LIN {X 0.075,Y -335.216,Z 1636.671,A 0.000,B 0.000,C 90.000,E1 120.797} C_DIS
LIN {X -0.094,Y -338.872,Z 1636.669,A 0.000,B 0.000,C 90.000,E1 120.384} C_DIS
LIN {X 0.042,Y -340.680,Z 1636.667,A 0.000,B 0.000,C 90.000,E1 120.050} C_DIS
LIN {X 0.186,Y -357.152,Z 1636.647,A 0.000,B 0.000,C 90.000,E1 116.360} C_DIS
LIN {X 0.077,Y -371.127,Z 1636.632,A 0.000,B 0.000,C 90.000,E1 113.695} C_DIS
LIN {X 0.128,Y -384.896,Z 1636.619,A 0.000,B 0.000,C 90.000,E1 111.354} C_DIS
LIN {X 0.030,Y -400.035,Z 1636.606,A 0.000,B 0.000,C 90.000,E1 109.087} C_DIS
LIN {X 0.035,Y -416.645,Z 1636.594,A 0.000,B 0.000,C 90.000,E1 106.858} C_DIS
LIN {X -0.200,Y -434.843,Z 1636.582,A 0.000,B 0.000,C 90.000,E1 104.717} C_DIS
LIN {X 0.091,Y -454.503,Z 1636.570,A 0.000,B 0.000,C 90.000,E1 102.591} C_DIS
LIN {X 0.158,Y -474.801,Z 1636.559,A 0.000,B 0.000,C 90.000,E1 100.658} C_DIS
LIN {X 0.135,Y -498.204,Z 1636.548,A 0.000,B 0.000,C 90.000,E1 98.681} C_DIS
LIN {X -0.215,Y -500.316,Z 1636.547,A 0.000,B 0.000,C 90.000,E1 98.511} C_DIS
LIN {X 0.233,Y -502.133,Z 1636.546,A 0.000,B 0.000,C 90.000,E1 98.219} C_DIS
LIN {X 0.114,Y -503.496,Z 1636.544,A 0.000,B 0.000,C 90.000,E1 97.992} C_DIS
LIN {X -0.087,Y -505.220,Z 1636.542,A 0.000,B 0.000,C 90.000,E1 97.530} C_DIS
LIN {X -0.279,Y -505.833,Z 1636.539,A 0.000,B 0.000,C 90.000,E1 97.068} C_DIS
LIN {X 0.041,Y -505.440,Z 1636.536,A 0.000,B 0.000,C 90.000,E1 96.549} C_DIS
LIN {X -0.139,Y -503.977,Z 1636.534,A 0.000,B 0.000,C 90.000,E1 96.087} C_DIS
LIN {X -0.204,Y -502.765,Z 1636.532,A 0.000,B 0.000,C 90.000,E1 95.853} C_DIS
LIN {X 0.120,Y -492.693,Z 1636.524,A 0.000,B 0.000,C 90.000,E1 94.359} C_DIS
LIN {X -0.215,Y -482.497,Z 1636.516,A 0.000,B 0.000,C 90.000,E1 92.922} C_DIS
LIN {X 0.208,Y -472.061,Z 1636.508,A 0.000,B 0.000,C 90.000,E1 91.375} C_DIS
LIN {X -0.031,Y -461.326,Z 1636.499,A 0.000,B 0.000,C 90.000,E1 89.885} C_DIS
LIN {X 0.010,Y -450.327,Z 1636.491,A 0.000,B 0.000,C 90.000,E1 88.339} C_DIS
LIN {X 0.132,Y -440.740,Z 1636.484,A 0.000,B 0.000,C 90.000,E1 87.020} C_DIS
LIN {X -0.147,Y -428.850,Z 1636.475,A 0.000,B 0.000,C 90.000,E1 85.469} C_DIS
LIN {X 0.070,Y -413.097,Z 1636.463,A 0.000,B 0.000,C 90.000,E1 83.280} C_DIS
LIN {X -0.188,Y -390.844,Z 1636.444,A 0.000,B 0.000,C 90.000,E1 79.982} C_DIS
LIN {X -0.184,Y -373.709,Z 1636.428,A 0.000,B 0.000,C 90.000,E1 77.117} C_DIS
LIN {X -0.093,Y -360.590,Z 1636.415,A 0.000,B 0.000,C 90.000,E1 74.755} C_DIS
LIN {X -0.182,Y -344.772,Z 1636.399,A 0.000,B 0.000,C 90.000,E1 71.764} C_DIS
LIN {X 0.065,Y -334.278,Z 1636.387,A 0.000,B 0.000,C 90.000,E1 69.571} C_DIS
LIN {X 0.131,Y -318.411,Z 1636.367,A 0.000,B 0.000,C 90.000,E1 66.102} C_DIS
LIN {X -0.065,Y -307.744,Z 1636.353,A 0.000,B 0.000,C 90.000,E1 63.563} C_DIS
LIN {X 0.008,Y -298.459,Z 1636.340,A 0.000,B 0.000,C 90.000,E1 61.257} C_DIS
LIN {X -0.096,Y -290.364,Z 1636.329,A 0.000,B 0.000,C 90.000,E1 59.282} C_DIS
LIN {X -0.050,Y -282.053,Z 1636.318,A 0.000,B 0.000,C 90.000,E1 57.248} C_DIS
LIN {X 0.091,Y -272.018,Z 1636.305,A 0.000,B 0.000,C 90.000,E1 54.815} C_DIS
LIN {X -0.053,Y -262.104,Z 1636.291,A 0.000,B 0.000,C 90.000,E1 52.396} C_DIS
LIN {X -0.034,Y -249.796,Z 1636.273,A 0.000,B 0.000,C 90.000,E1 49.175} C_DIS
LIN {X -0.085,Y -238.241,Z 1636.255,A 0.000,B 0.000,C 90.000,E1 45.891} C_DIS
LIN {X -0.115,Y -227.562,Z 1636.236,A 0.000,B 0.000,C 90.000,E1 42.528} C_DIS
LIN {X 0.011,Y -218.837,Z 1636.219,A 0.000,B 0.000,C 90.000,E1 39.439} C_DIS
LIN {X 0.134,Y -210.840,Z 1636.202,A 0.000,B 0.000,C 90.000,E1 36.297} C_DIS
LIN {X 0.025,Y -203.747,Z 1636.184,A 0.000,B 0.000,C 90.000,E1 33.166} C_DIS
LIN {X 0.042,Y -197.376,Z 1636.167,A 0.000,B 0.000,C 90.000,E1 29.951} C_DIS
LIN {X 0.054,Y -191.738,Z 1636.148,A 0.000,B 0.000,C 90.000,E1 26.693} C_DIS
LIN {X 0.092,Y -186.712,Z 1636.130,A 0.000,B 0.000,C 90.000,E1 23.387} C_DIS
LIN {X 0.054,Y -182.428,Z 1636.112,A 0.000,B 0.000,C 90.000,E1 20.066} C_DIS
LIN {X -0.074,Y -177.974,Z 1636.088,A 0.000,B 0.000,C 90.000,E1 15.898} C_DIS
LIN {X 0.065,Y -174.306,Z 1636.065,A 0.000,B 0.000,C 90.000,E1 11.602} C_DIS
LIN {X -0.026,Y -171.007,Z 1636.036,A 0.000,B 0.000,C 90.000,E1 6.486} C_DIS
LIN {X -0.031,Y -168.517,Z 1635.997,A 0.000,B 0.000,C 90.000,E1 359.542} C_DIS
LIN {X 0.016,Y -168.866,Z 1635.939,A 0.000,B 0.000,C 90.000,E1 349.106} C_DIS
LIN {X -0.013,Y -171.390,Z 1635.911,A 0.000,B 0.000,C 90.000,E1 343.921} C_DIS
LIN {X -0.035,Y -174.661,Z 1635.887,A 0.000,B 0.000,C 90.000,E1 339.625} C_DIS
LIN {X 0.059,Y -178.265,Z 1635.868,A 0.000,B 0.000,C 90.000,E1 336.177} C_DIS
LIN {X 0.044,Y -182.804,Z 1635.849,A 0.000,B 0.000,C 90.000,E1 332.794} C_DIS
LIN {X -0.010,Y -188.198,Z 1635.830,A 0.000,B 0.000,C 90.000,E1 329.459} C_DIS
LIN {X 0.034,Y -194.339,Z 1635.812,A 0.000,B 0.000,C 90.000,E1 326.135} C_DIS
LIN {X -0.030,Y -201.410,Z 1635.794,A 0.000,B 0.000,C 90.000,E1 322.889} C_DIS
LIN {X -0.008,Y -208.249,Z 1635.778,A 0.000,B 0.000,C 90.000,E1 320.070} C_DIS
LIN {X 0.019,Y -217.241,Z 1635.761,A 0.000,B 0.000,C 90.000,E1 316.905} C_DIS
LIN {X 0.119,Y -227.424,Z 1635.743,A 0.000,B 0.000,C 90.000,E1 313.785} C_DIS
LIN {X 0.049,Y -237.290,Z 1635.729,A 0.000,B 0.000,C 90.000,E1 311.148} C_DIS
LIN {X 0.078,Y -246.746,Z 1635.716,A 0.000,B 0.000,C 90.000,E1 308.910} C_DIS
LIN {X -0.018,Y -257.358,Z 1635.704,A 0.000,B 0.000,C 90.000,E1 306.744} C_DIS
LIN {X -0.070,Y -269.099,Z 1635.692,A 0.000,B 0.000,C 90.000,E1 304.612} C_DIS
LIN {X 0.026,Y -281.970,Z 1635.681,A 0.000,B 0.000,C 90.000,E1 302.498} C_DIS
LIN {X -0.013,Y -303.406,Z 1635.664,A 0.000,B 0.000,C 90.000,E1 299.461} C_DIS
LIN {X -0.163,Y -315.909,Z 1635.655,A 0.000,B 0.000,C 90.000,E1 297.847} C_DIS
LIN {X -0.021,Y -330.723,Z 1635.644,A 0.000,B 0.000,C 90.000,E1 295.899} C_DIS
LIN {X -0.018,Y -342.793,Z 1635.635,A 0.000,B 0.000,C 90.000,E1 294.335} C_DIS
LIN {X -0.111,Y -357.187,Z 1635.625,A 0.000,B 0.000,C 90.000,E1 292.514} C_DIS
LIN {X 0.176,Y -369.073,Z 1635.617,A 0.000,B 0.000,C 90.000,E1 290.972} C_DIS
LIN {X 0.069,Y -378.254,Z 1635.610,A 0.000,B 0.000,C 90.000,E1 289.812} C_DIS
LIN {X -0.059,Y -384.632,Z 1635.605,A 0.000,B 0.000,C 90.000,E1 288.960} C_DIS
LIN {X 0.232,Y -390.479,Z 1635.600,A 0.000,B 0.000,C 90.000,E1 288.055} C_DIS
LIN {X 0.095,Y -395.675,Z 1635.596,A 0.000,B 0.000,C 90.000,E1 287.221} C_DIS
LIN {X 0.002,Y -400.090,Z 1635.591,A 0.000,B 0.000,C 90.000,E1 286.386} C_DIS
LIN {X -0.046,Y -403.619,Z 1635.586,A 0.000,B 0.000,C 90.000,E1 285.552} C_DIS
LIN {X -0.066,Y -406.336,Z 1635.582,A 0.000,B 0.000,C 90.000,E1 284.717} C_DIS
LIN {X 0.227,Y -407.692,Z 1635.579,A 0.000,B 0.000,C 90.000,E1 284.120} C_DIS
LIN {X 0.033,Y -408.625,Z 1635.576,A 0.000,B 0.000,C 90.000,E1 283.592} C_DIS
LIN {X -0.151,Y -409.111,Z 1635.573,A 0.000,B 0.000,C 90.000,E1 283.063} C_DIS
LIN {X 0.071,Y -409.049,Z 1635.569,A 0.000,B 0.000,C 90.000,E1 282.479} C_DIS
LIN {X -0.104,Y -408.553,Z 1635.566,A 0.000,B 0.000,C 90.000,E1 281.951} C_DIS
LIN {X 0.122,Y -407.464,Z 1635.563,A 0.000,B 0.000,C 90.000,E1 281.366} C_DIS
LIN {X -0.056,Y -405.832,Z 1635.560,A 0.000,B 0.000,C 90.000,E1 280.838} C_DIS
LIN {X 0.155,Y -403.556,Z 1635.557,A 0.000,B 0.000,C 90.000,E1 280.254} C_DIS
LIN {X -0.048,Y -400.589,Z 1635.554,A 0.000,B 0.000,C 90.000,E1 279.726} C_DIS
LIN {X 0.062,Y -396.918,Z 1635.551,A 0.000,B 0.000,C 90.000,E1 279.151} C_DIS
LIN {X -0.166,Y -390.492,Z 1635.546,A 0.000,B 0.000,C 90.000,E1 278.341} C_DIS
LIN {X -0.006,Y -383.215,Z 1635.542,A 0.000,B 0.000,C 90.000,E1 277.466} C_DIS
LIN {X 0.010,Y -377.815,Z 1635.538,A 0.000,B 0.000,C 90.000,E1 276.891} C_DIS
LIN {X -0.157,Y -372.074,Z 1635.535,A 0.000,B 0.000,C 90.000,E1 276.372} C_DIS
LIN {X -0.088,Y -366.074,Z 1635.532,A 0.000,B 0.000,C 90.000,E1 275.853} C_DIS
LIN {X -0.143,Y -359.715,Z 1635.530,A 0.000,B 0.000,C 90.000,E1 275.391} C_DIS
LIN {X 0.085,Y -353.409,Z 1635.527,A 0.000,B 0.000,C 90.000,E1 274.935} C_DIS
LIN {X -0.164,Y -343.745,Z 1635.524,A 0.000,B 0.000,C 90.000,E1 274.416} C_DIS
LIN {X -0.072,Y -333.992,Z 1635.522,A 0.000,B 0.000,C 90.000,E1 273.898} C_DIS
LIN {X 0.044,Y -324.586,Z 1635.519,A 0.000,B 0.000,C 90.000,E1 273.440} C_DIS
LIN {X 0.029,Y -314.581,Z 1635.517,A 0.000,B 0.000,C 90.000,E1 273.037} C_DIS
LIN {X 0.023,Y -304.485,Z 1635.515,A 0.000,B 0.000,C 90.000,E1 272.694} C_DIS
LIN {X 0.017,Y -293.887,Z 1635.513,A 0.000,B 0.000,C 90.000,E1 272.407} C_DIS
LIN {X 0.055,Y -286.273,Z 1635.512,A 0.000,B 0.000,C 90.000,E1 272.236} C_DIS
LIN {X -0.068,Y -277.615,Z 1635.512,A 0.000,B 0.000,C 90.000,E1 272.121} C_DIS
LIN {X 0.043,Y -254.563,Z 1635.511,A 0.000,B 0.000,C 90.000,E1 271.892} C_DIS
LIN {X 0.074,Y -223.653,Z 1635.509,A 0.000,B 0.000,C 90.000,E1 271.661} C_DIS
LIN {X 0.057,Y -206.714,Z 1635.509,A 0.000,B 0.000,C 90.000,E1 271.604} C_DIS
LIN {X 0.032,Y -199.398,Z 1635.509,A 0.000,B 0.000,C 90.000,E1 271.604} C_DIS
LIN {X -0.014,Y -191.538,Z 1635.509,A 0.000,B 0.000,C 90.000,E1 271.604} C_DIS
LIN {X -0.034,Y -181.333,Z 1635.509,A 0.000,B 0.000,C 90.000,E1 271.604} C_DIS
LIN {X 0.027,Y -181.569,Z 1635.500,A 0.000,B 0.000,C 90.000,E1 270.057} C_DIS
LIN {X -0.016,Y -180.905,Z 1635.474,A 0.000,B 0.000,C 90.000,E1 265.355} C_DIS
LIN {X 0.058,Y -180.679,Z 1635.469,A 0.000,B 0.000,C 90.000,E1 264.489} C_DIS
LIN {X -0.044,Y -178.761,Z 1635.441,A 0.000,B 0.000,C 90.000,E1 259.454} C_DIS
LIN {X 0.029,Y -175.809,Z 1635.413,A 0.000,B 0.000,C 90.000,E1 254.338} C_DIS
LIN {X 0.023,Y -171.995,Z 1635.385,A 0.000,B 0.000,C 90.000,E1 249.209} C_DIS
LIN {X -0.003,Y -171.407,Z 1635.380,A 0.000,B 0.000,C 90.000,E1 248.358} C_DIS
LIN {X 0.045,Y -167.647,Z 1635.356,A 0.000,B 0.000,C 90.000,E1 244.024} C_DIS
LIN {X 0.060,Y -166.310,Z 1635.346,A 0.000,B 0.000,C 90.000,E1 242.281} C_DIS
LIN {X 0.054,Y -163.053,Z 1635.327,A 0.000,B 0.000,C 90.000,E1 238.791} C_DIS
LIN {X 0.015,Y -160.988,Z 1635.312,A 0.000,B 0.000,C 90.000,E1 236.167} C_DIS
LIN {X -0.007,Y -157.736,Z 1635.292,A 0.000,B 0.000,C 90.000,E1 232.637} C_DIS
LIN {X -0.069,Y -155.775,Z 1635.278,A 0.000,B 0.000,C 90.000,E1 229.989} C_DIS
LIN {X -0.014,Y -152.030,Z 1635.253,A 0.000,B 0.000,C 90.000,E1 225.486} C_DIS
LIN {X 0.004,Y -150.278,Z 1635.238,A 0.000,B 0.000,C 90.000,E1 222.771} C_DIS
LIN {X 0.022,Y -147.028,Z 1635.212,A 0.000,B 0.000,C 90.000,E1 218.222} C_DIS
LIN {X -0.077,Y -145.609,Z 1635.197,A 0.000,B 0.000,C 90.000,E1 215.518} C_DIS
LIN {X 0.046,Y -142.995,Z 1635.172,A 0.000,B 0.000,C 90.000,E1 210.875} C_DIS
LIN {X -0.019,Y -141.622,Z 1635.151,A 0.000,B 0.000,C 90.000,E1 207.206} C_DIS
LIN {X 0.037,Y -139.431,Z 1635.115,A 0.000,B 0.000,C 90.000,E1 200.684} C_DIS
LIN {X -0.040,Y -139.162,Z 1635.105,A 0.000,B 0.000,C 90.000,E1 198.852} C_DIS
LIN {X -0.003,Y -138.341,Z 1635.058,A 0.000,B 0.000,C 90.000,E1 190.433} C_DIS
LIN {X 0.005,Y -139.478,Z 1635.006,A 0.000,B 0.000,C 90.000,E1 181.088} C_DIS
LIN {X -0.055,Y -141.064,Z 1634.975,A 0.000,B 0.000,C 90.000,E1 175.527} C_DIS
LIN {X 0.040,Y -142.438,Z 1634.960,A 0.000,B 0.000,C 90.000,E1 172.704} C_DIS
LIN {X -0.041,Y -144.677,Z 1634.934,A 0.000,B 0.000,C 90.000,E1 168.117} C_DIS
LIN {X -0.057,Y -147.265,Z 1634.913,A 0.000,B 0.000,C 90.000,E1 164.448} C_DIS
LIN {X -0.040,Y -150.583,Z 1634.888,A 0.000,B 0.000,C 90.000,E1 159.880} C_DIS
LIN {X 0.039,Y -154.054,Z 1634.868,A 0.000,B 0.000,C 90.000,E1 156.230} C_DIS
LIN {X -0.035,Y -157.473,Z 1634.848,A 0.000,B 0.000,C 90.000,E1 152.666} C_DIS
LIN {X 0.052,Y -161.695,Z 1634.828,A 0.000,B 0.000,C 90.000,E1 149.076} C_DIS
LIN {X -0.071,Y -165.889,Z 1634.809,A 0.000,B 0.000,C 90.000,E1 145.595} C_DIS
LIN {X 0.054,Y -170.871,Z 1634.789,A 0.000,B 0.000,C 90.000,E1 142.065} C_DIS
LIN {X -0.034,Y -175.740,Z 1634.770,A 0.000,B 0.000,C 90.000,E1 138.647} C_DIS
LIN {X -0.044,Y -181.350,Z 1634.751,A 0.000,B 0.000,C 90.000,E1 135.243} C_DIS
LIN {X 0.089,Y -186.840,Z 1634.733,A 0.000,B 0.000,C 90.000,E1 131.838} C_DIS
LIN {X 0.043,Y -191.427,Z 1634.719,A 0.000,B 0.000,C 90.000,E1 129.358} C_DIS
LIN {X -0.025,Y -197.278,Z 1634.700,A 0.000,B 0.000,C 90.000,E1 126.091} C_DIS
LIN {X 0.012,Y -200.555,Z 1634.691,A 0.000,B 0.000,C 90.000,E1 124.452} C_DIS
LIN {X 0.126,Y -206.322,Z 1634.674,A 0.000,B 0.000,C 90.000,E1 121.258} C_DIS
LIN {X 0.163,Y -325.904,Z 1634.674,A 0.000,B 0.000,C 90.000,E1 121.258} C_DIS
LIN {X -0.138,Y -328.739,Z 1634.674,A 0.000,B 0.000,C 90.000,E1 121.258} C_DIS
LIN {X 0.066,Y -331.867,Z 1634.673,A 0.000,B 0.000,C 90.000,E1 121.082} C_DIS
LIN {X 0.096,Y -335.415,Z 1634.671,A 0.000,B 0.000,C 90.000,E1 120.797} C_DIS
LIN {X 0.116,Y -339.039,Z 1634.669,A 0.000,B 0.000,C 90.000,E1 120.335} C_DIS
LIN {X -0.041,Y -340.765,Z 1634.667,A 0.000,B 0.000,C 90.000,E1 120.050} C_DIS
LIN {X 0.063,Y -355.738,Z 1634.648,A 0.000,B 0.000,C 90.000,E1 116.668} C_DIS
LIN {X -0.092,Y -369.545,Z 1634.633,A 0.000,B 0.000,C 90.000,E1 114.003} C_DIS
LIN {X -0.090,Y -383.157,Z 1634.620,A 0.000,B 0.000,C 90.000,E1 111.663} C_DIS
LIN {X -0.237,Y -398.126,Z 1634.608,A 0.000,B 0.000,C 90.000,E1 109.396} C_DIS
LIN {X 0.232,Y -414.554,Z 1634.595,A 0.000,B 0.000,C 90.000,E1 107.094} C_DIS
LIN {X -0.046,Y -432.555,Z 1634.583,A 0.000,B 0.000,C 90.000,E1 104.954} C_DIS
LIN {X 0.135,Y -452.080,Z 1634.571,A 0.000,B 0.000,C 90.000,E1 102.827} C_DIS
LIN {X 0.044,Y -472.312,Z 1634.561,A 0.000,B 0.000,C 90.000,E1 100.894} C_DIS
LIN {X 0.048,Y -498.275,Z 1634.548,A 0.000,B 0.000,C 90.000,E1 98.681} C_DIS
LIN {X 0.192,Y -500.325,Z 1634.547,A 0.000,B 0.000,C 90.000,E1 98.454} C_DIS
LIN {X 0.117,Y -502.115,Z 1634.546,A 0.000,B 0.000,C 90.000,E1 98.219} C_DIS
LIN {X -0.030,Y -503.453,Z 1634.544,A 0.000,B 0.000,C 90.000,E1 97.992} C_DIS
LIN {X -0.230,Y -505.107,Z 1634.542,A 0.000,B 0.000,C 90.000,E1 97.530} C_DIS
LIN {X 0.140,Y -505.662,Z 1634.539,A 0.000,B 0.000,C 90.000,E1 97.004} C_DIS
LIN {X -0.104,Y -505.211,Z 1634.536,A 0.000,B 0.000,C 90.000,E1 96.549} C_DIS
LIN {X 0.217,Y -503.682,Z 1634.534,A 0.000,B 0.000,C 90.000,E1 96.030} C_DIS
LIN {X 0.150,Y -502.429,Z 1634.532,A 0.000,B 0.000,C 90.000,E1 95.796} C_DIS
LIN {X -0.165,Y -490.665,Z 1634.523,A 0.000,B 0.000,C 90.000,E1 94.131} C_DIS
LIN {X -0.044,Y -480.435,Z 1634.515,A 0.000,B 0.000,C 90.000,E1 92.636} C_DIS
LIN {X -0.128,Y -469.962,Z 1634.506,A 0.000,B 0.000,C 90.000,E1 91.146} C_DIS
LIN {X 0.066,Y -459.199,Z 1634.498,A 0.000,B 0.000,C 90.000,E1 89.599} C_DIS
LIN {X -0.147,Y -450.009,Z 1634.491,A 0.000,B 0.000,C 90.000,E1 88.339} C_DIS
LIN {X -0.026,Y -440.399,Z 1634.483,A 0.000,B 0.000,C 90.000,E1 87.020} C_DIS
LIN {X 0.120,Y -428.487,Z 1634.475,A 0.000,B 0.000,C 90.000,E1 85.412} C_DIS
LIN {X -0.019,Y -410.774,Z 1634.461,A 0.000,B 0.000,C 90.000,E1 82.996} C_DIS
LIN {X 0.086,Y -388.715,Z 1634.443,A 0.000,B 0.000,C 90.000,E1 79.634} C_DIS
LIN {X 0.096,Y -371.677,Z 1634.427,A 0.000,B 0.000,C 90.000,E1 76.756} C_DIS
LIN {X 0.137,Y -358.613,Z 1634.413,A 0.000,B 0.000,C 90.000,E1 74.393} C_DIS
LIN {X -0.002,Y -341.412,Z 1634.395,A 0.000,B 0.000,C 90.000,E1 71.094} C_DIS
LIN {X 0.170,Y -330.932,Z 1634.383,A 0.000,B 0.000,C 90.000,E1 68.901} C_DIS
LIN {X -0.051,Y -318.060,Z 1634.367,A 0.000,B 0.000,C 90.000,E1 66.102} C_DIS
LIN {X 0.028,Y -307.443,Z 1634.353,A 0.000,B 0.000,C 90.000,E1 63.512} C_DIS
LIN {X -0.176,Y -298.201,Z 1634.340,A 0.000,B 0.000,C 90.000,E1 61.257} C_DIS
LIN {X 0.118,Y -290.106,Z 1634.329,A 0.000,B 0.000,C 90.000,E1 59.203} C_DIS
LIN {X 0.004,Y -281.799,Z 1634.318,A 0.000,B 0.000,C 90.000,E1 57.199} C_DIS
LIN {X 0.035,Y -273.191,Z 1634.306,A 0.000,B 0.000,C 90.000,E1 55.135} C_DIS
LIN {X 0.072,Y -263.226,Z 1634.293,A 0.000,B 0.000,C 90.000,E1 52.683} C_DIS
LIN {X 0.090,Y -252.129,Z 1634.277,A 0.000,B 0.000,C 90.000,E1 49.828} C_DIS
LIN {X 0.115,Y -240.407,Z 1634.259,A 0.000,B 0.000,C 90.000,E1 46.539} C_DIS
LIN {X -0.033,Y -229.500,Z 1634.240,A 0.000,B 0.000,C 90.000,E1 43.218} C_DIS
LIN {X -0.039,Y -220.614,Z 1634.223,A 0.000,B 0.000,C 90.000,E1 40.172} C_DIS
LIN {X -0.039,Y -212.488,Z 1634.206,A 0.000,B 0.000,C 90.000,E1 37.076} C_DIS
LIN {X 0.012,Y -205.212,Z 1634.188,A 0.000,B 0.000,C 90.000,E1 33.913} C_DIS
LIN {X -0.005,Y -198.723,Z 1634.171,A 0.000,B 0.000,C 90.000,E1 30.718} C_DIS
LIN {X 0.034,Y -192.949,Z 1634.153,A 0.000,B 0.000,C 90.000,E1 27.462} C_DIS
LIN {X -0.067,Y -187.805,Z 1634.134,A 0.000,B 0.000,C 90.000,E1 24.207} C_DIS
LIN {X -0.005,Y -183.406,Z 1634.116,A 0.000,B 0.000,C 90.000,E1 20.865} C_DIS
LIN {X -0.044,Y -178.803,Z 1634.093,A 0.000,B 0.000,C 90.000,E1 16.677} C_DIS
LIN {X 0.029,Y -174.999,Z 1634.069,A 0.000,B 0.000,C 90.000,E1 12.411} C_DIS
LIN {X -0.042,Y -171.514,Z 1634.040,A 0.000,B 0.000,C 90.000,E1 7.296} C_DIS
LIN {X -0.081,Y -168.833,Z 1634.002,A 0.000,B 0.000,C 90.000,E1 0.401} C_DIS
LIN {X 0.025,Y -169.007,Z 1633.940,A 0.000,B 0.000,C 90.000,E1 349.106} C_DIS
LIN {X 0.001,Y -171.541,Z 1633.911,A 0.000,B 0.000,C 90.000,E1 343.921} C_DIS
LIN {X -0.016,Y -174.815,Z 1633.887,A 0.000,B 0.000,C 90.000,E1 339.625} C_DIS
LIN {X -0.081,Y -178.413,Z 1633.868,A 0.000,B 0.000,C 90.000,E1 336.230} C_DIS
LIN {X -0.012,Y -182.957,Z 1633.849,A 0.000,B 0.000,C 90.000,E1 332.820} C_DIS
LIN {X 0.022,Y -188.363,Z 1633.830,A 0.000,B 0.000,C 90.000,E1 329.459} C_DIS
LIN {X -0.036,Y -194.515,Z 1633.812,A 0.000,B 0.000,C 90.000,E1 326.167} C_DIS
LIN {X -0.108,Y -201.568,Z 1633.794,A 0.000,B 0.000,C 90.000,E1 322.924} C_DIS
LIN {X 0.040,Y -208.410,Z 1633.778,A 0.000,B 0.000,C 90.000,E1 320.070} C_DIS
LIN {X 0.074,Y -217.363,Z 1633.761,A 0.000,B 0.000,C 90.000,E1 316.905} C_DIS
LIN {X 0.090,Y -226.182,Z 1633.746,A 0.000,B 0.000,C 90.000,E1 314.190} C_DIS
LIN {X 0.114,Y -237.349,Z 1633.729,A 0.000,B 0.000,C 90.000,E1 311.148} C_DIS
LIN {X -0.046,Y -246.761,Z 1633.716,A 0.000,B 0.000,C 90.000,E1 308.955} C_DIS
LIN {X 0.053,Y -257.345,Z 1633.704,A 0.000,B 0.000,C 90.000,E1 306.744} C_DIS
LIN {X 0.004,Y -269.072,Z 1633.692,A 0.000,B 0.000,C 90.000,E1 304.612} C_DIS
LIN {X -0.134,Y -281.926,Z 1633.681,A 0.000,B 0.000,C 90.000,E1 302.546} C_DIS
LIN {X 0.070,Y -303.397,Z 1633.664,A 0.000,B 0.000,C 90.000,E1 299.461} C_DIS
LIN {X -0.077,Y -315.881,Z 1633.655,A 0.000,B 0.000,C 90.000,E1 297.847} C_DIS
LIN {X -0.076,Y -330.696,Z 1633.644,A 0.000,B 0.000,C 90.000,E1 295.924} C_DIS
LIN {X 0.075,Y -342.761,Z 1633.635,A 0.000,B 0.000,C 90.000,E1 294.335} C_DIS
LIN {X -0.013,Y -357.126,Z 1633.625,A 0.000,B 0.000,C 90.000,E1 292.514} C_DIS
LIN {X -0.200,Y -369.005,Z 1633.617,A 0.000,B 0.000,C 90.000,E1 291.046} C_DIS
LIN {X 0.171,Y -378.226,Z 1633.610,A 0.000,B 0.000,C 90.000,E1 289.812} C_DIS
LIN {X 0.045,Y -384.631,Z 1633.605,A 0.000,B 0.000,C 90.000,E1 288.960} C_DIS
LIN {X -0.155,Y -390.471,Z 1633.601,A 0.000,B 0.000,C 90.000,E1 288.127} C_DIS
LIN {X -0.176,Y -395.717,Z 1633.596,A 0.000,B 0.000,C 90.000,E1 287.275} C_DIS
LIN {X 0.049,Y -398.795,Z 1633.593,A 0.000,B 0.000,C 90.000,E1 286.677} C_DIS
LIN {X -0.018,Y -402.648,Z 1633.588,A 0.000,B 0.000,C 90.000,E1 285.843} C_DIS
LIN {X -0.135,Y -404.748,Z 1633.585,A 0.000,B 0.000,C 90.000,E1 285.300} C_DIS
LIN {X 0.046,Y -406.503,Z 1633.582,A 0.000,B 0.000,C 90.000,E1 284.717} C_DIS
LIN {X -0.055,Y -407.888,Z 1633.579,A 0.000,B 0.000,C 90.000,E1 284.175} C_DIS
LIN {X 0.149,Y -408.876,Z 1633.576,A 0.000,B 0.000,C 90.000,E1 283.592} C_DIS
LIN {X -0.035,Y -409.392,Z 1633.573,A 0.000,B 0.000,C 90.000,E1 283.063} C_DIS
LIN {X -0.212,Y -409.414,Z 1633.569,A 0.000,B 0.000,C 90.000,E1 282.535} C_DIS
LIN {X 0.016,Y -408.919,Z 1633.566,A 0.000,B 0.000,C 90.000,E1 281.951} C_DIS
LIN {X -0.157,Y -407.877,Z 1633.563,A 0.000,B 0.000,C 90.000,E1 281.422} C_DIS
LIN {X 0.067,Y -406.293,Z 1633.560,A 0.000,B 0.000,C 90.000,E1 280.838} C_DIS
LIN {X -0.117,Y -404.031,Z 1633.557,A 0.000,B 0.000,C 90.000,E1 280.310} C_DIS
LIN {X 0.079,Y -401.109,Z 1633.554,A 0.000,B 0.000,C 90.000,E1 279.726} C_DIS
LIN {X -0.200,Y -397.535,Z 1633.551,A 0.000,B 0.000,C 90.000,E1 279.208} C_DIS
LIN {X -0.035,Y -391.127,Z 1633.546,A 0.000,B 0.000,C 90.000,E1 278.341} C_DIS
LIN {X 0.079,Y -383.768,Z 1633.542,A 0.000,B 0.000,C 90.000,E1 277.473} C_DIS
LIN {X 0.172,Y -378.343,Z 1633.538,A 0.000,B 0.000,C 90.000,E1 276.891} C_DIS
LIN {X 0.055,Y -372.695,Z 1633.535,A 0.000,B 0.000,C 90.000,E1 276.372} C_DIS
LIN {X 0.139,Y -366.713,Z 1633.533,A 0.000,B 0.000,C 90.000,E1 275.853} C_DIS
LIN {X 0.107,Y -360.444,Z 1633.530,A 0.000,B 0.000,C 90.000,E1 275.391} C_DIS
LIN {X -0.057,Y -354.071,Z 1633.528,A 0.000,B 0.000,C 90.000,E1 274.992} C_DIS
LIN {X 0.059,Y -347.600,Z 1633.526,A 0.000,B 0.000,C 90.000,E1 274.588} C_DIS
LIN {X 0.052,Y -337.974,Z 1633.523,A 0.000,B 0.000,C 90.000,E1 274.073} C_DIS
LIN {X 0.039,Y -328.302,Z 1633.520,A 0.000,B 0.000,C 90.000,E1 273.612} C_DIS
LIN {X -0.017,Y -318.764,Z 1633.518,A 0.000,B 0.000,C 90.000,E1 273.212} C_DIS
LIN {X 0.139,Y -308.410,Z 1633.516,A 0.000,B 0.000,C 90.000,E1 272.808} C_DIS
LIN {X 0.024,Y -298.197,Z 1633.514,A 0.000,B 0.000,C 90.000,E1 272.522} C_DIS
LIN {X -0.110,Y -286.864,Z 1633.513,A 0.000,B 0.000,C 90.000,E1 272.293} C_DIS
LIN {X 0.045,Y -278.334,Z 1633.512,A 0.000,B 0.000,C 90.000,E1 272.121} C_DIS
LIN {X 0.075,Y -261.202,Z 1633.511,A 0.000,B 0.000,C 90.000,E1 271.949} C_DIS
LIN {X 0.000,Y -229.135,Z 1633.510,A 0.000,B 0.000,C 90.000,E1 271.718} C_DIS
LIN {X -0.086,Y -210.090,Z 1633.509,A 0.000,B 0.000,C 90.000,E1 271.661} C_DIS
LIN {X 0.083,Y -204.360,Z 1633.509,A 0.000,B 0.000,C 90.000,E1 271.604} C_DIS
LIN {X 0.041,Y -181.329,Z 1633.509,A 0.000,B 0.000,C 90.000,E1 271.604} C_DIS
LIN {X -0.015,Y -181.538,Z 1633.499,A 0.000,B 0.000,C 90.000,E1 269.885} C_DIS
LIN {X -0.031,Y -180.813,Z 1633.471,A 0.000,B 0.000,C 90.000,E1 264.837} C_DIS
LIN {X 0.046,Y -178.916,Z 1633.443,A 0.000,B 0.000,C 90.000,E1 259.746} C_DIS
LIN {X -0.044,Y -175.962,Z 1633.415,A 0.000,B 0.000,C 90.000,E1 254.685} C_DIS
LIN {X 0.071,Y -175.436,Z 1633.410,A 0.000,B 0.000,C 90.000,E1 253.795} C_DIS
LIN {X 0.074,Y -172.194,Z 1633.386,A 0.000,B 0.000,C 90.000,E1 249.518} C_DIS
LIN {X 0.050,Y -171.667,Z 1633.382,A 0.000,B 0.000,C 90.000,E1 248.666} C_DIS
LIN {X 0.034,Y -167.892,Z 1633.358,A 0.000,B 0.000,C 90.000,E1 244.357} C_DIS
LIN {X 0.049,Y -166.631,Z 1633.348,A 0.000,B 0.000,C 90.000,E1 242.615} C_DIS
LIN {X 0.043,Y -162.616,Z 1633.324,A 0.000,B 0.000,C 90.000,E1 238.250} C_DIS
LIN {X 0.016,Y -161.302,Z 1633.314,A 0.000,B 0.000,C 90.000,E1 236.501} C_DIS
LIN {X 0.050,Y -157.300,Z 1633.289,A 0.000,B 0.000,C 90.000,E1 232.065} C_DIS
LIN {X 0.078,Y -155.276,Z 1633.275,A 0.000,B 0.000,C 90.000,E1 229.380} C_DIS
LIN {X 0.007,Y -151.642,Z 1633.250,A 0.000,B 0.000,C 90.000,E1 224.919} C_DIS
LIN {X 0.054,Y -150.510,Z 1633.240,A 0.000,B 0.000,C 90.000,E1 223.095} C_DIS
LIN {X -0.032,Y -147.235,Z 1633.214,A 0.000,B 0.000,C 90.000,E1 218.588} C_DIS
LIN {X 0.052,Y -145.259,Z 1633.194,A 0.000,B 0.000,C 90.000,E1 214.898} C_DIS
LIN {X -0.032,Y -142.371,Z 1633.163,A 0.000,B 0.000,C 90.000,E1 209.411} C_DIS
LIN {X -0.037,Y -141.756,Z 1633.153,A 0.000,B 0.000,C 90.000,E1 207.564} C_DIS
LIN {X 0.014,Y -139.496,Z 1633.117,A 0.000,B 0.000,C 90.000,E1 201.046} C_DIS
LIN {X 0.051,Y -139.003,Z 1633.101,A 0.000,B 0.000,C 90.000,E1 198.236} C_DIS
LIN {X 0.008,Y -138.339,Z 1633.055,A 0.000,B 0.000,C 90.000,E1 189.849} C_DIS
LIN {X 0.030,Y -139.407,Z 1633.008,A 0.000,B 0.000,C 90.000,E1 181.432} C_DIS
LIN {X -0.057,Y -141.317,Z 1632.972,A 0.000,B 0.000,C 90.000,E1 174.951} C_DIS
LIN {X 0.042,Y -142.676,Z 1632.956,A 0.000,B 0.000,C 90.000,E1 172.129} C_DIS
LIN {X 0.021,Y -145.030,Z 1632.931,A 0.000,B 0.000,C 90.000,E1 167.521} C_DIS
LIN {X -0.022,Y -147.657,Z 1632.910,A 0.000,B 0.000,C 90.000,E1 163.866} C_DIS
LIN {X 0.055,Y -150.294,Z 1632.890,A 0.000,B 0.000,C 90.000,E1 160.188} C_DIS
LIN {X -0.075,Y -153.702,Z 1632.870,A 0.000,B 0.000,C 90.000,E1 156.613} C_DIS
LIN {X -0.020,Y -157.115,Z 1632.850,A 0.000,B 0.000,C 90.000,E1 152.999} C_DIS
LIN {X 0.057,Y -161.258,Z 1632.830,A 0.000,B 0.000,C 90.000,E1 149.410} C_DIS
LIN {X -0.015,Y -164.377,Z 1632.815,A 0.000,B 0.000,C 90.000,E1 146.786} C_DIS
LIN {X -0.029,Y -169.051,Z 1632.796,A 0.000,B 0.000,C 90.000,E1 143.290} C_DIS
LIN {X 0.024,Y -171.612,Z 1632.786,A 0.000,B 0.000,C 90.000,E1 141.537} C_DIS
LIN {X 0.072,Y -176.569,Z 1632.767,A 0.000,B 0.000,C 90.000,E1 138.081} C_DIS
LIN {X -0.055,Y -180.867,Z 1632.753,A 0.000,B 0.000,C 90.000,E1 135.567} C_DIS
LIN {X 0.067,Y -186.280,Z 1632.734,A 0.000,B 0.000,C 90.000,E1 132.162} C_DIS
LIN {X -0.012,Y -190.915,Z 1632.720,A 0.000,B 0.000,C 90.000,E1 129.688} C_DIS
LIN {X 0.055,Y -196.682,Z 1632.702,A 0.000,B 0.000,C 90.000,E1 126.377} C_DIS
LIN {X 0.087,Y -199.925,Z 1632.693,A 0.000,B 0.000,C 90.000,E1 124.739} C_DIS
LIN {X 0.004,Y -204.317,Z 1632.680,A 0.000,B 0.000,C 90.000,E1 122.339} C_DIS
LIN {X 0.004,Y -206.234,Z 1632.674,A 0.000,B 0.000,C 90.000,E1 121.337} C_DIS
LIN {X -0.030,Y -325.247,Z 1632.674,A 0.000,B 0.000,C 90.000,E1 121.337} C_DIS
LIN {X 0.059,Y -327.773,Z 1632.674,A 0.000,B 0.000,C 90.000,E1 121.288} C_DIS
LIN {X 0.089,Y -333.375,Z 1632.672,A 0.000,B 0.000,C 90.000,E1 121.003} C_DIS
LIN {X 0.117,Y -336.315,Z 1632.671,A 0.000,B 0.000,C 90.000,E1 120.718} C_DIS
LIN {X -0.009,Y -339.955,Z 1632.668,A 0.000,B 0.000,C 90.000,E1 120.207} C_DIS
LIN {X -0.025,Y -342.716,Z 1632.664,A 0.000,B 0.000,C 90.000,E1 119.589} C_DIS
LIN {X 0.087,Y -354.962,Z 1632.649,A 0.000,B 0.000,C 90.000,E1 116.821} C_DIS
LIN {X 0.072,Y -368.683,Z 1632.634,A 0.000,B 0.000,C 90.000,E1 114.131} C_DIS
LIN {X 0.060,Y -382.211,Z 1632.621,A 0.000,B 0.000,C 90.000,E1 111.791} C_DIS
LIN {X 0.030,Y -397.089,Z 1632.608,A 0.000,B 0.000,C 90.000,E1 109.504} C_DIS
LIN {X -0.043,Y -413.418,Z 1632.596,A 0.000,B 0.000,C 90.000,E1 107.275} C_DIS
LIN {X 0.167,Y -431.315,Z 1632.584,A 0.000,B 0.000,C 90.000,E1 105.064} C_DIS
LIN {X -0.255,Y -450.769,Z 1632.572,A 0.000,B 0.000,C 90.000,E1 103.008} C_DIS
LIN {X 0.107,Y -470.966,Z 1632.561,A 0.000,B 0.000,C 90.000,E1 101.007} C_DIS
LIN {X -0.182,Y -494.291,Z 1632.550,A 0.000,B 0.000,C 90.000,E1 99.029} C_DIS
LIN {X 0.157,Y -499.269,Z 1632.548,A 0.000,B 0.000,C 90.000,E1 98.568} C_DIS
LIN {X -0.184,Y -501.036,Z 1632.547,A 0.000,B 0.000,C 90.000,E1 98.398} C_DIS
LIN {X 0.240,Y -502.602,Z 1632.545,A 0.000,B 0.000,C 90.000,E1 98.106} C_DIS
LIN {X 0.167,Y -503.769,Z 1632.544,A 0.000,B 0.000,C 90.000,E1 97.871} C_DIS
LIN {X -0.034,Y -505.154,Z 1632.541,A 0.000,B 0.000,C 90.000,E1 97.409} C_DIS
LIN {X -0.229,Y -505.479,Z 1632.538,A 0.000,B 0.000,C 90.000,E1 96.947} C_DIS
LIN {X 0.087,Y -504.796,Z 1632.536,A 0.000,B 0.000,C 90.000,E1 96.429} C_DIS
LIN {X -0.098,Y -502.993,Z 1632.533,A 0.000,B 0.000,C 90.000,E1 95.967} C_DIS
LIN {X -0.217,Y -501.561,Z 1632.532,A 0.000,B 0.000,C 90.000,E1 95.739} C_DIS
LIN {X -0.161,Y -488.067,Z 1632.521,A 0.000,B 0.000,C 90.000,E1 93.784} C_DIS
LIN {X -0.114,Y -477.778,Z 1632.513,A 0.000,B 0.000,C 90.000,E1 92.293} C_DIS
LIN {X 0.227,Y -467.247,Z 1632.504,A 0.000,B 0.000,C 90.000,E1 90.745} C_DIS
LIN {X -0.088,Y -456.463,Z 1632.496,A 0.000,B 0.000,C 90.000,E1 89.255} C_DIS
LIN {X 0.129,Y -447.133,Z 1632.489,A 0.000,B 0.000,C 90.000,E1 87.936} C_DIS
LIN {X 0.203,Y -437.387,Z 1632.481,A 0.000,B 0.000,C 90.000,E1 86.617} C_DIS
LIN {X 0.001,Y -423.469,Z 1632.471,A 0.000,B 0.000,C 90.000,E1 84.780} C_DIS
LIN {X -0.100,Y -404.050,Z 1632.456,A 0.000,B 0.000,C 90.000,E1 82.064} C_DIS
LIN {X -0.210,Y -382.545,Z 1632.437,A 0.000,B 0.000,C 90.000,E1 78.701} C_DIS
LIN {X 0.075,Y -365.838,Z 1632.421,A 0.000,B 0.000,C 90.000,E1 75.755} C_DIS
LIN {X 0.068,Y -352.899,Z 1632.408,A 0.000,B 0.000,C 90.000,E1 73.378} C_DIS
LIN {X -0.144,Y -337.569,Z 1632.391,A 0.000,B 0.000,C 90.000,E1 70.369} C_DIS
LIN {X -0.005,Y -324.216,Z 1632.375,A 0.000,B 0.000,C 90.000,E1 67.539} C_DIS
LIN {X -0.014,Y -309.337,Z 1632.356,A 0.000,B 0.000,C 90.000,E1 64.024} C_DIS
LIN {X 0.112,Y -298.817,Z 1632.341,A 0.000,B 0.000,C 90.000,E1 61.385} C_DIS
LIN {X 0.013,Y -290.758,Z 1632.330,A 0.000,B 0.000,C 90.000,E1 59.410} C_DIS
LIN {X 0.065,Y -282.494,Z 1632.319,A 0.000,B 0.000,C 90.000,E1 57.375} C_DIS
LIN {X 0.115,Y -273.878,Z 1632.307,A 0.000,B 0.000,C 90.000,E1 55.308} C_DIS
LIN {X 0.011,Y -263.890,Z 1632.294,A 0.000,B 0.000,C 90.000,E1 52.889} C_DIS
LIN {X -0.111,Y -252.693,Z 1632.278,A 0.000,B 0.000,C 90.000,E1 50.070} C_DIS
LIN {X -0.062,Y -240.893,Z 1632.260,A 0.000,B 0.000,C 90.000,E1 46.782} C_DIS
LIN {X -0.026,Y -229.909,Z 1632.241,A 0.000,B 0.000,C 90.000,E1 43.419} C_DIS
LIN {X -0.098,Y -219.951,Z 1632.222,A 0.000,B 0.000,C 90.000,E1 40.011} C_DIS
LIN {X 0.054,Y -211.899,Z 1632.205,A 0.000,B 0.000,C 90.000,E1 36.870} C_DIS
LIN {X 0.089,Y -204.706,Z 1632.187,A 0.000,B 0.000,C 90.000,E1 33.706} C_DIS
LIN {X -0.044,Y -198.303,Z 1632.170,A 0.000,B 0.000,C 90.000,E1 30.541} C_DIS
LIN {X 0.081,Y -192.581,Z 1632.152,A 0.000,B 0.000,C 90.000,E1 27.257} C_DIS
LIN {X -0.035,Y -187.532,Z 1632.133,A 0.000,B 0.000,C 90.000,E1 24.003} C_DIS
LIN {X 0.013,Y -183.215,Z 1632.115,A 0.000,B 0.000,C 90.000,E1 20.663} C_DIS
LIN {X 0.075,Y -178.674,Z 1632.091,A 0.000,B 0.000,C 90.000,E1 16.441} C_DIS
LIN {X -0.065,Y -174.928,Z 1632.068,A 0.000,B 0.000,C 90.000,E1 12.243} C_DIS
LIN {X 0.042,Y -171.518,Z 1632.039,A 0.000,B 0.000,C 90.000,E1 7.068} C_DIS
LIN {X 0.000,Y -168.866,Z 1632.000,A 0.000,B 0.000,C 90.000,E1 360.000} C_DIS
LIN {X 0.035,Y -169.150,Z 1631.940,A 0.000,B 0.000,C 90.000,E1 349.106} C_DIS
LIN {X 0.016,Y -171.692,Z 1631.911,A 0.000,B 0.000,C 90.000,E1 343.921} C_DIS
LIN {X 0.004,Y -174.970,Z 1631.887,A 0.000,B 0.000,C 90.000,E1 339.625} C_DIS
LIN {X -0.057,Y -178.568,Z 1631.868,A 0.000,B 0.000,C 90.000,E1 336.230} C_DIS
LIN {X 0.017,Y -183.124,Z 1631.849,A 0.000,B 0.000,C 90.000,E1 332.820} C_DIS
LIN {X 0.056,Y -188.528,Z 1631.830,A 0.000,B 0.000,C 90.000,E1 329.459} C_DIS
LIN {X 0.002,Y -194.695,Z 1631.812,A 0.000,B 0.000,C 90.000,E1 326.167} C_DIS
LIN {X -0.063,Y -201.727,Z 1631.794,A 0.000,B 0.000,C 90.000,E1 322.924} C_DIS
LIN {X -0.024,Y -209.611,Z 1631.776,A 0.000,B 0.000,C 90.000,E1 319.703} C_DIS
LIN {X -0.018,Y -217.484,Z 1631.761,A 0.000,B 0.000,C 90.000,E1 316.944} C_DIS
LIN {X -0.010,Y -226.267,Z 1631.746,A 0.000,B 0.000,C 90.000,E1 314.231} C_DIS
LIN {X 0.002,Y -237.391,Z 1631.729,A 0.000,B 0.000,C 90.000,E1 311.191} C_DIS
LIN {X 0.024,Y -246.773,Z 1631.716,A 0.000,B 0.000,C 90.000,E1 308.955} C_DIS
LIN {X -0.081,Y -257.320,Z 1631.704,A 0.000,B 0.000,C 90.000,E1 306.790} C_DIS
LIN {X -0.006,Y -271.092,Z 1631.690,A 0.000,B 0.000,C 90.000,E1 304.278} C_DIS
LIN {X -0.104,Y -284.152,Z 1631.679,A 0.000,B 0.000,C 90.000,E1 302.212} C_DIS
LIN {X 0.004,Y -303.370,Z 1631.664,A 0.000,B 0.000,C 90.000,E1 299.489} C_DIS
LIN {X 0.009,Y -315.845,Z 1631.655,A 0.000,B 0.000,C 90.000,E1 297.847} C_DIS
LIN {X 0.014,Y -330.667,Z 1631.644,A 0.000,B 0.000,C 90.000,E1 295.924} C_DIS
LIN {X -0.145,Y -342.719,Z 1631.635,A 0.000,B 0.000,C 90.000,E1 294.387} C_DIS
LIN {X 0.080,Y -357.075,Z 1631.625,A 0.000,B 0.000,C 90.000,E1 292.514} C_DIS
LIN {X -0.020,Y -371.306,Z 1631.615,A 0.000,B 0.000,C 90.000,E1 290.737} C_DIS
LIN {X -0.088,Y -378.242,Z 1631.610,A 0.000,B 0.000,C 90.000,E1 289.866} C_DIS
LIN {X 0.143,Y -384.629,Z 1631.605,A 0.000,B 0.000,C 90.000,E1 288.960} C_DIS
LIN {X -0.056,Y -390.501,Z 1631.601,A 0.000,B 0.000,C 90.000,E1 288.127} C_DIS
LIN {X -0.075,Y -395.793,Z 1631.596,A 0.000,B 0.000,C 90.000,E1 287.275} C_DIS
LIN {X -0.171,Y -400.274,Z 1631.591,A 0.000,B 0.000,C 90.000,E1 286.441} C_DIS
LIN {X -0.221,Y -403.889,Z 1631.587,A 0.000,B 0.000,C 90.000,E1 285.607} C_DIS
LIN {X 0.153,Y -406.687,Z 1631.582,A 0.000,B 0.000,C 90.000,E1 284.717} C_DIS
LIN {X 0.052,Y -408.087,Z 1631.579,A 0.000,B 0.000,C 90.000,E1 284.175} C_DIS
LIN {X -0.141,Y -409.147,Z 1631.576,A 0.000,B 0.000,C 90.000,E1 283.647} C_DIS
LIN {X 0.075,Y -409.661,Z 1631.573,A 0.000,B 0.000,C 90.000,E1 283.063} C_DIS
LIN {X -0.100,Y -409.765,Z 1631.570,A 0.000,B 0.000,C 90.000,E1 282.535} C_DIS
LIN {X 0.129,Y -409.279,Z 1631.567,A 0.000,B 0.000,C 90.000,E1 281.951} C_DIS
LIN {X -0.042,Y -408.344,Z 1631.563,A 0.000,B 0.000,C 90.000,E1 281.422} C_DIS
LIN {X 0.182,Y -406.745,Z 1631.560,A 0.000,B 0.000,C 90.000,E1 280.838} C_DIS
LIN {X 0.002,Y -404.530,Z 1631.557,A 0.000,B 0.000,C 90.000,E1 280.310} C_DIS
LIN {X 0.200,Y -401.678,Z 1631.554,A 0.000,B 0.000,C 90.000,E1 279.726} C_DIS
LIN {X -0.078,Y -398.138,Z 1631.551,A 0.000,B 0.000,C 90.000,E1 279.208} C_DIS
LIN {X 0.091,Y -391.760,Z 1631.546,A 0.000,B 0.000,C 90.000,E1 278.341} C_DIS
LIN {X -0.173,Y -384.360,Z 1631.542,A 0.000,B 0.000,C 90.000,E1 277.530} C_DIS
LIN {X -0.048,Y -378.941,Z 1631.539,A 0.000,B 0.000,C 90.000,E1 276.947} C_DIS
LIN {X -0.170,Y -373.229,Z 1631.536,A 0.000,B 0.000,C 90.000,E1 276.429} C_DIS
LIN {X -0.057,Y -367.259,Z 1631.533,A 0.000,B 0.000,C 90.000,E1 275.910} C_DIS
LIN {X -0.070,Y -361.112,Z 1631.530,A 0.000,B 0.000,C 90.000,E1 275.454} C_DIS
LIN {X 0.143,Y -354.756,Z 1631.528,A 0.000,B 0.000,C 90.000,E1 274.992} C_DIS
LIN {X -0.117,Y -348.218,Z 1631.526,A 0.000,B 0.000,C 90.000,E1 274.645} C_DIS
LIN {X -0.113,Y -338.574,Z 1631.523,A 0.000,B 0.000,C 90.000,E1 274.131} C_DIS
LIN {X -0.127,Y -328.866,Z 1631.520,A 0.000,B 0.000,C 90.000,E1 273.669} C_DIS
LIN {X 0.106,Y -319.112,Z 1631.518,A 0.000,B 0.000,C 90.000,E1 273.212} C_DIS
LIN {X -0.056,Y -308.903,Z 1631.516,A 0.000,B 0.000,C 90.000,E1 272.865} C_DIS
LIN {X -0.003,Y -301.868,Z 1631.515,A 0.000,B 0.000,C 90.000,E1 272.636} C_DIS
LIN {X 0.054,Y -290.778,Z 1631.513,A 0.000,B 0.000,C 90.000,E1 272.350} C_DIS
LIN {X -0.135,Y -282.707,Z 1631.512,A 0.000,B 0.000,C 90.000,E1 272.236} C_DIS
LIN {X 0.082,Y -266.959,Z 1631.511,A 0.000,B 0.000,C 90.000,E1 272.007} C_DIS
LIN {X 0.031,Y -229.173,Z 1631.510,A 0.000,B 0.000,C 90.000,E1 271.718} C_DIS
LIN {X -0.059,Y -209.081,Z 1631.509,A 0.000,B 0.000,C 90.000,E1 271.661} C_DIS
LIN {X -0.086,Y -181.326,Z 1631.509,A 0.000,B 0.000,C 90.000,E1 271.661} C_DIS
LIN {X -0.008,Y -181.538,Z 1631.499,A 0.000,B 0.000,C 90.000,E1 269.885} C_DIS
LIN {X -0.024,Y -180.815,Z 1631.471,A 0.000,B 0.000,C 90.000,E1 264.837} C_DIS
LIN {X 0.053,Y -178.917,Z 1631.443,A 0.000,B 0.000,C 90.000,E1 259.746} C_DIS
LIN {X -0.037,Y -175.962,Z 1631.415,A 0.000,B 0.000,C 90.000,E1 254.685} C_DIS
LIN {X 0.079,Y -175.438,Z 1631.410,A 0.000,B 0.000,C 90.000,E1 253.795} C_DIS
LIN {X -0.080,Y -172.196,Z 1631.386,A 0.000,B 0.000,C 90.000,E1 249.571} C_DIS
LIN {X -0.102,Y -171.669,Z 1631.382,A 0.000,B 0.000,C 90.000,E1 248.720} C_DIS
LIN {X 0.040,Y -167.894,Z 1631.358,A 0.000,B 0.000,C 90.000,E1 244.357} C_DIS
LIN {X 0.056,Y -166.633,Z 1631.348,A 0.000,B 0.000,C 90.000,E1 242.615} C_DIS
LIN {X -0.037,Y -162.618,Z 1631.324,A 0.000,B 0.000,C 90.000,E1 238.280} C_DIS
LIN {X 0.023,Y -161.304,Z 1631.314,A 0.000,B 0.000,C 90.000,E1 236.501} C_DIS
LIN {X -0.068,Y -157.301,Z 1631.289,A 0.000,B 0.000,C 90.000,E1 232.110} C_DIS
LIN {X 0.085,Y -155.278,Z 1631.275,A 0.000,B 0.000,C 90.000,E1 229.380} C_DIS
LIN {X 0.014,Y -151.643,Z 1631.250,A 0.000,B 0.000,C 90.000,E1 224.919} C_DIS
LIN {X -0.050,Y -150.512,Z 1631.240,A 0.000,B 0.000,C 90.000,E1 223.137} C_DIS
LIN {X -0.026,Y -147.236,Z 1631.214,A 0.000,B 0.000,C 90.000,E1 218.588} C_DIS
LIN {X 0.058,Y -145.260,Z 1631.194,A 0.000,B 0.000,C 90.000,E1 214.898} C_DIS
LIN {X -0.026,Y -142.372,Z 1631.163,A 0.000,B 0.000,C 90.000,E1 209.411} C_DIS
LIN {X -0.031,Y -141.757,Z 1631.153,A 0.000,B 0.000,C 90.000,E1 207.564} C_DIS
LIN {X 0.020,Y -139.497,Z 1631.117,A 0.000,B 0.000,C 90.000,E1 201.046} C_DIS
LIN {X 0.057,Y -139.003,Z 1631.101,A 0.000,B 0.000,C 90.000,E1 198.236} C_DIS
LIN {X 0.014,Y -138.339,Z 1631.055,A 0.000,B 0.000,C 90.000,E1 189.849} C_DIS
LIN {X 0.036,Y -139.407,Z 1631.008,A 0.000,B 0.000,C 90.000,E1 181.432} C_DIS
LIN {X -0.051,Y -141.316,Z 1630.972,A 0.000,B 0.000,C 90.000,E1 174.951} C_DIS
LIN {X 0.048,Y -142.676,Z 1630.956,A 0.000,B 0.000,C 90.000,E1 172.129} C_DIS
LIN {X 0.028,Y -145.028,Z 1630.931,A 0.000,B 0.000,C 90.000,E1 167.521} C_DIS
LIN {X -0.015,Y -147.655,Z 1630.910,A 0.000,B 0.000,C 90.000,E1 163.866} C_DIS
LIN {X 0.061,Y -150.292,Z 1630.890,A 0.000,B 0.000,C 90.000,E1 160.188} C_DIS
LIN {X -0.068,Y -153.699,Z 1630.870,A 0.000,B 0.000,C 90.000,E1 156.613} C_DIS
LIN {X -0.013,Y -157.113,Z 1630.850,A 0.000,B 0.000,C 90.000,E1 152.999} C_DIS
LIN {X 0.063,Y -161.255,Z 1630.830,A 0.000,B 0.000,C 90.000,E1 149.410} C_DIS
LIN {X -0.009,Y -164.374,Z 1630.815,A 0.000,B 0.000,C 90.000,E1 146.786} C_DIS
LIN {X -0.021,Y -169.048,Z 1630.796,A 0.000,B 0.000,C 90.000,E1 143.290} C_DIS
LIN {X 0.031,Y -171.609,Z 1630.786,A 0.000,B 0.000,C 90.000,E1 141.537} C_DIS
LIN {X 0.079,Y -176.565,Z 1630.767,A 0.000,B 0.000,C 90.000,E1 138.081} C_DIS
LIN {X -0.048,Y -180.863,Z 1630.753,A 0.000,B 0.000,C 90.000,E1 135.567} C_DIS
LIN {X -0.063,Y -186.276,Z 1630.734,A 0.000,B 0.000,C 90.000,E1 132.204} C_DIS
LIN {X -0.005,Y -190.911,Z 1630.720,A 0.000,B 0.000,C 90.000,E1 129.688} C_DIS
LIN {X 0.063,Y -196.678,Z 1630.702,A 0.000,B 0.000,C 90.000,E1 126.377} C_DIS
LIN {X -0.019,Y -199.921,Z 1630.693,A 0.000,B 0.000,C 90.000,E1 124.771} C_DIS
LIN {X 0.011,Y -204.312,Z 1630.680,A 0.000,B 0.000,C 90.000,E1 122.339} C_DIS
LIN {X -0.035,Y -206.158,Z 1630.674,A 0.000,B 0.000,C 90.000,E1 121.386} C_DIS
LIN {X -0.104,Y -326.119,Z 1630.674,A 0.000,B 0.000,C 90.000,E1 121.386} C_DIS
LIN {X -0.029,Y -331.028,Z 1630.673,A 0.000,B 0.000,C 90.000,E1 121.209} C_DIS
LIN {X -0.014,Y -333.325,Z 1630.672,A 0.000,B 0.000,C 90.000,E1 121.052} C_DIS
LIN {X -0.042,Y -336.467,Z 1630.671,A 0.000,B 0.000,C 90.000,E1 120.747} C_DIS
LIN {X -0.077,Y -340.042,Z 1630.668,A 0.000,B 0.000,C 90.000,E1 120.207} C_DIS
LIN {X 0.217,Y -346.667,Z 1630.659,A 0.000,B 0.000,C 90.000,E1 118.615} C_DIS
LIN {X -0.027,Y -359.399,Z 1630.644,A 0.000,B 0.000,C 90.000,E1 115.924} C_DIS
LIN {X -0.073,Y -373.641,Z 1630.629,A 0.000,B 0.000,C 90.000,E1 113.259} C_DIS
LIN {X 0.038,Y -387.669,Z 1630.616,A 0.000,B 0.000,C 90.000,E1 110.918} C_DIS
LIN {X -0.131,Y -403.084,Z 1630.604,A 0.000,B 0.000,C 90.000,E1 108.671} C_DIS
LIN {X -0.052,Y -419.995,Z 1630.591,A 0.000,B 0.000,C 90.000,E1 106.441} C_DIS
LIN {X -0.210,Y -438.516,Z 1630.579,A 0.000,B 0.000,C 90.000,E1 104.300} C_DIS
LIN {X -0.231,Y -458.334,Z 1630.568,A 0.000,B 0.000,C 90.000,E1 102.243} C_DIS
LIN {X 0.085,Y -478.735,Z 1630.557,A 0.000,B 0.000,C 90.000,E1 100.310} C_DIS
LIN {X -0.143,Y -497.008,Z 1630.549,A 0.000,B 0.000,C 90.000,E1 98.803} C_DIS
LIN {X 0.085,Y -499.284,Z 1630.548,A 0.000,B 0.000,C 90.000,E1 98.568} C_DIS
LIN {X -0.256,Y -501.008,Z 1630.547,A 0.000,B 0.000,C 90.000,E1 98.398} C_DIS
LIN {X 0.168,Y -502.540,Z 1630.545,A 0.000,B 0.000,C 90.000,E1 98.106} C_DIS
LIN {X 0.094,Y -503.679,Z 1630.544,A 0.000,B 0.000,C 90.000,E1 97.871} C_DIS
LIN {X -0.107,Y -505.021,Z 1630.541,A 0.000,B 0.000,C 90.000,E1 97.409} C_DIS
LIN {X 0.200,Y -505.307,Z 1630.538,A 0.000,B 0.000,C 90.000,E1 96.891} C_DIS
LIN {X 0.013,Y -504.584,Z 1630.536,A 0.000,B 0.000,C 90.000,E1 96.429} C_DIS
LIN {X -0.172,Y -502.733,Z 1630.533,A 0.000,B 0.000,C 90.000,E1 95.967} C_DIS
LIN {X 0.089,Y -499.564,Z 1630.530,A 0.000,B 0.000,C 90.000,E1 95.454} C_DIS
LIN {X 0.100,Y -486.087,Z 1630.520,A 0.000,B 0.000,C 90.000,E1 93.498} C_DIS
LIN {X -0.051,Y -474.057,Z 1630.510,A 0.000,B 0.000,C 90.000,E1 91.776} C_DIS
LIN {X 0.210,Y -463.429,Z 1630.501,A 0.000,B 0.000,C 90.000,E1 90.229} C_DIS
LIN {X 0.060,Y -454.399,Z 1630.494,A 0.000,B 0.000,C 90.000,E1 88.969} C_DIS
LIN {X -0.207,Y -444.922,Z 1630.487,A 0.000,B 0.000,C 90.000,E1 87.707} C_DIS
LIN {X 0.003,Y -433.141,Z 1630.478,A 0.000,B 0.000,C 90.000,E1 86.102} C_DIS
LIN {X -0.103,Y -417.210,Z 1630.466,A 0.000,B 0.000,C 90.000,E1 83.970} C_DIS
LIN {X 0.113,Y -396.338,Z 1630.450,A 0.000,B 0.000,C 90.000,E1 80.905} C_DIS
LIN {X 0.201,Y -378.837,Z 1630.434,A 0.000,B 0.000,C 90.000,E1 78.049} C_DIS
LIN {X -0.054,Y -363.898,Z 1630.419,A 0.000,B 0.000,C 90.000,E1 75.463} C_DIS
LIN {X -0.108,Y -351.032,Z 1630.406,A 0.000,B 0.000,C 90.000,E1 73.087} C_DIS
LIN {X 0.053,Y -335.761,Z 1630.389,A 0.000,B 0.000,C 90.000,E1 70.007} C_DIS
LIN {X 0.036,Y -319.728,Z 1630.370,A 0.000,B 0.000,C 90.000,E1 66.561} C_DIS
LIN {X -0.091,Y -307.763,Z 1630.354,A 0.000,B 0.000,C 90.000,E1 63.691} C_DIS
LIN {X -0.012,Y -298.595,Z 1630.341,A 0.000,B 0.000,C 90.000,E1 61.385} C_DIS
LIN {X -0.111,Y -290.553,Z 1630.330,A 0.000,B 0.000,C 90.000,E1 59.410} C_DIS
LIN {X -0.059,Y -282.297,Z 1630.319,A 0.000,B 0.000,C 90.000,E1 57.375} C_DIS
LIN {X -0.008,Y -273.677,Z 1630.307,A 0.000,B 0.000,C 90.000,E1 55.308} C_DIS
LIN {X 0.096,Y -263.667,Z 1630.294,A 0.000,B 0.000,C 90.000,E1 52.844} C_DIS
LIN {X 0.119,Y -252.398,Z 1630.278,A 0.000,B 0.000,C 90.000,E1 49.989} C_DIS
LIN {X -0.024,Y -240.566,Z 1630.260,A 0.000,B 0.000,C 90.000,E1 46.743} C_DIS
LIN {X 0.002,Y -229.613,Z 1630.241,A 0.000,B 0.000,C 90.000,E1 43.380} C_DIS
LIN {X 0.079,Y -219.681,Z 1630.222,A 0.000,B 0.000,C 90.000,E1 39.930} C_DIS
LIN {X -0.079,Y -211.686,Z 1630.205,A 0.000,B 0.000,C 90.000,E1 36.870} C_DIS
LIN {X -0.045,Y -204.533,Z 1630.187,A 0.000,B 0.000,C 90.000,E1 33.706} C_DIS
LIN {X 0.093,Y -198.167,Z 1630.169,A 0.000,B 0.000,C 90.000,E1 30.463} C_DIS
LIN {X -0.052,Y -192.481,Z 1630.151,A 0.000,B 0.000,C 90.000,E1 27.257} C_DIS
LIN {X 0.004,Y -187.495,Z 1630.133,A 0.000,B 0.000,C 90.000,E1 23.951} C_DIS
LIN {X 0.054,Y -183.209,Z 1630.115,A 0.000,B 0.000,C 90.000,E1 20.610} C_DIS
LIN {X -0.052,Y -178.713,Z 1630.091,A 0.000,B 0.000,C 90.000,E1 16.441} C_DIS
LIN {X -0.017,Y -174.983,Z 1630.068,A 0.000,B 0.000,C 90.000,E1 12.187} C_DIS
LIN {X 0.093,Y -172.075,Z 1630.044,A 0.000,B 0.000,C 90.000,E1 7.871} C_DIS
LIN {X -0.074,Y -169.500,Z 1630.010,A 0.000,B 0.000,C 90.000,E1 1.892} C_DIS
LIN {X -0.062,Y -169.983,Z 1629.930,A 0.000,B 0.000,C 90.000,E1 347.409} C_DIS
LIN {X 0.083,Y -173.020,Z 1629.901,A 0.000,B 0.000,C 90.000,E1 342.181} C_DIS
LIN {X 0.003,Y -176.796,Z 1629.877,A 0.000,B 0.000,C 90.000,E1 337.922} C_DIS
LIN {X -0.043,Y -180.877,Z 1629.859,A 0.000,B 0.000,C 90.000,E1 334.537} C_DIS
LIN {X -0.076,Y -185.905,Z 1629.840,A 0.000,B 0.000,C 90.000,E1 331.179} C_DIS
LIN {X -0.031,Y -191.670,Z 1629.821,A 0.000,B 0.000,C 90.000,E1 327.837} C_DIS
LIN {X -0.066,Y -198.299,Z 1629.803,A 0.000,B 0.000,C 90.000,E1 324.562} C_DIS
LIN {X -0.086,Y -205.704,Z 1629.785,A 0.000,B 0.000,C 90.000,E1 321.331} C_DIS
LIN {X -0.015,Y -213.028,Z 1629.770,A 0.000,B 0.000,C 90.000,E1 318.528} C_DIS
LIN {X -0.021,Y -222.475,Z 1629.752,A 0.000,B 0.000,C 90.000,E1 315.405} C_DIS
LIN {X -0.111,Y -233.122,Z 1629.735,A 0.000,B 0.000,C 90.000,E1 312.366} C_DIS
LIN {X -0.016,Y -241.946,Z 1629.723,A 0.000,B 0.000,C 90.000,E1 310.092} C_DIS
LIN {X -0.064,Y -250.158,Z 1629.712,A 0.000,B 0.000,C 90.000,E1 308.257} C_DIS
LIN {X -0.101,Y -261.059,Z 1629.700,A 0.000,B 0.000,C 90.000,E1 306.091} C_DIS
LIN {X 0.064,Y -275.233,Z 1629.687,A 0.000,B 0.000,C 90.000,E1 303.579} C_DIS
LIN {X -0.072,Y -286.420,Z 1629.677,A 0.000,B 0.000,C 90.000,E1 301.878} C_DIS
LIN {X 0.100,Y -305.844,Z 1629.662,A 0.000,B 0.000,C 90.000,E1 299.155} C_DIS
LIN {X 0.154,Y -318.256,Z 1629.653,A 0.000,B 0.000,C 90.000,E1 297.513} C_DIS
LIN {X -0.093,Y -333.039,Z 1629.642,A 0.000,B 0.000,C 90.000,E1 295.643} C_DIS
LIN {X -0.063,Y -345.054,Z 1629.634,A 0.000,B 0.000,C 90.000,E1 294.079} C_DIS
LIN {X 0.213,Y -359.408,Z 1629.624,A 0.000,B 0.000,C 90.000,E1 292.206} C_DIS
LIN {X 0.163,Y -373.615,Z 1629.614,A 0.000,B 0.000,C 90.000,E1 290.429} C_DIS
LIN {X -0.003,Y -380.377,Z 1629.609,A 0.000,B 0.000,C 90.000,E1 289.577} C_DIS
LIN {X -0.118,Y -386.655,Z 1629.604,A 0.000,B 0.000,C 90.000,E1 288.725} C_DIS
LIN {X 0.201,Y -392.374,Z 1629.599,A 0.000,B 0.000,C 90.000,E1 287.819} C_DIS
LIN {X 0.077,Y -397.421,Z 1629.594,A 0.000,B 0.000,C 90.000,E1 286.985} C_DIS
LIN {X -0.067,Y -400.371,Z 1629.591,A 0.000,B 0.000,C 90.000,E1 286.441} C_DIS
LIN {X -0.115,Y -404.017,Z 1629.587,A 0.000,B 0.000,C 90.000,E1 285.607} C_DIS
LIN {X -0.134,Y -406.882,Z 1629.582,A 0.000,B 0.000,C 90.000,E1 284.773} C_DIS
LIN {X 0.061,Y -408.330,Z 1629.579,A 0.000,B 0.000,C 90.000,E1 284.189} C_DIS
LIN {X -0.030,Y -409.363,Z 1629.576,A 0.000,B 0.000,C 90.000,E1 283.647} C_DIS
LIN {X 0.187,Y -409.952,Z 1629.573,A 0.000,B 0.000,C 90.000,E1 283.063} C_DIS
LIN {X 0.014,Y -410.016,Z 1629.570,A 0.000,B 0.000,C 90.000,E1 282.535} C_DIS
LIN {X -0.157,Y -409.631,Z 1629.567,A 0.000,B 0.000,C 90.000,E1 282.007} C_DIS
LIN {X 0.073,Y -408.778,Z 1629.563,A 0.000,B 0.000,C 90.000,E1 281.422} C_DIS
LIN {X -0.099,Y -407.181,Z 1629.560,A 0.000,B 0.000,C 90.000,E1 280.894} C_DIS
LIN {X 0.121,Y -405.048,Z 1629.557,A 0.000,B 0.000,C 90.000,E1 280.310} C_DIS
LIN {X -0.137,Y -402.245,Z 1629.554,A 0.000,B 0.000,C 90.000,E1 279.792} C_DIS
LIN {X 0.050,Y -398.736,Z 1629.551,A 0.000,B 0.000,C 90.000,E1 279.208} C_DIS
LIN {X 0.213,Y -394.645,Z 1629.548,A 0.000,B 0.000,C 90.000,E1 278.624} C_DIS
LIN {X -0.040,Y -387.592,Z 1629.543,A 0.000,B 0.000,C 90.000,E1 277.814} C_DIS
LIN {X 0.011,Y -382.296,Z 1629.540,A 0.000,B 0.000,C 90.000,E1 277.239} C_DIS
LIN {X 0.155,Y -376.676,Z 1629.537,A 0.000,B 0.000,C 90.000,E1 276.663} C_DIS
LIN {X 0.144,Y -370.838,Z 1629.534,A 0.000,B 0.000,C 90.000,E1 276.144} C_DIS
LIN {X 0.034,Y -364.697,Z 1629.532,A 0.000,B 0.000,C 90.000,E1 275.682} C_DIS
LIN {X 0.168,Y -358.449,Z 1629.529,A 0.000,B 0.000,C 90.000,E1 275.220} C_DIS
LIN {X -0.181,Y -352.156,Z 1629.527,A 0.000,B 0.000,C 90.000,E1 274.878} C_DIS
LIN {X 0.034,Y -342.459,Z 1629.524,A 0.000,B 0.000,C 90.000,E1 274.302} C_DIS
LIN {X -0.055,Y -332.833,Z 1629.521,A 0.000,B 0.000,C 90.000,E1 273.841} C_DIS
LIN {X 0.066,Y -323.072,Z 1629.519,A 0.000,B 0.000,C 90.000,E1 273.383} C_DIS
LIN {X -0.143,Y -313.194,Z 1629.517,A 0.000,B 0.000,C 90.000,E1 273.037} C_DIS
LIN {X -0.134,Y -302.778,Z 1629.515,A 0.000,B 0.000,C 90.000,E1 272.694} C_DIS
LIN {X 0.034,Y -295.346,Z 1629.514,A 0.000,B 0.000,C 90.000,E1 272.465} C_DIS
LIN {X -0.013,Y -283.605,Z 1629.512,A 0.000,B 0.000,C 90.000,E1 272.236} C_DIS
LIN {X -0.077,Y -268.386,Z 1629.511,A 0.000,B 0.000,C 90.000,E1 272.064} C_DIS
LIN {X 0.001,Y -235.035,Z 1629.510,A 0.000,B 0.000,C 90.000,E1 271.776} C_DIS
LIN {X 0.001,Y -213.573,Z 1629.509,A 0.000,B 0.000,C 90.000,E1 271.661} C_DIS
LIN {X -0.038,Y -207.614,Z 1629.509,A 0.000,B 0.000,C 90.000,E1 271.661} C_DIS
LIN {X -0.068,Y -181.324,Z 1629.509,A 0.000,B 0.000,C 90.000,E1 271.661} C_DIS
LIN {X 0.084,Y -181.545,Z 1629.500,A 0.000,B 0.000,C 90.000,E1 269.885} C_DIS
LIN {X 0.067,Y -180.824,Z 1629.471,A 0.000,B 0.000,C 90.000,E1 264.837} C_DIS
LIN {X -0.033,Y -178.928,Z 1629.443,A 0.000,B 0.000,C 90.000,E1 259.803} C_DIS
LIN {X 0.006,Y -175.976,Z 1629.415,A 0.000,B 0.000,C 90.000,E1 254.700} C_DIS
LIN {X -0.049,Y -175.463,Z 1629.410,A 0.000,B 0.000,C 90.000,E1 253.866} C_DIS
LIN {X 0.008,Y -172.214,Z 1629.386,A 0.000,B 0.000,C 90.000,E1 249.571} C_DIS
LIN {X -0.014,Y -171.689,Z 1629.382,A 0.000,B 0.000,C 90.000,E1 248.720} C_DIS
LIN {X -0.024,Y -167.916,Z 1629.358,A 0.000,B 0.000,C 90.000,E1 244.409} C_DIS
LIN {X -0.005,Y -166.658,Z 1629.348,A 0.000,B 0.000,C 90.000,E1 242.666} C_DIS
LIN {X 0.049,Y -162.641,Z 1629.324,A 0.000,B 0.000,C 90.000,E1 238.280} C_DIS
LIN {X -0.027,Y -161.330,Z 1629.314,A 0.000,B 0.000,C 90.000,E1 236.548} C_DIS
LIN {X 0.017,Y -157.325,Z 1629.290,A 0.000,B 0.000,C 90.000,E1 232.110} C_DIS
LIN {X -0.051,Y -155.307,Z 1629.275,A 0.000,B 0.000,C 90.000,E1 229.461} C_DIS
LIN {X -0.012,Y -151.664,Z 1629.250,A 0.000,B 0.000,C 90.000,E1 224.960} C_DIS
LIN {X 0.032,Y -150.530,Z 1629.240,A 0.000,B 0.000,C 90.000,E1 223.137} C_DIS
LIN {X -0.037,Y -147.256,Z 1629.214,A 0.000,B 0.000,C 90.000,E1 218.624} C_DIS
LIN {X 0.020,Y -145.281,Z 1629.194,A 0.000,B 0.000,C 90.000,E1 214.945} C_DIS
LIN {X 0.053,Y -142.383,Z 1629.163,A 0.000,B 0.000,C 90.000,E1 209.411} C_DIS
LIN {X -0.024,Y -141.361,Z 1629.148,A 0.000,B 0.000,C 90.000,E1 206.668} C_DIS
LIN {X -0.046,Y -139.343,Z 1629.112,A 0.000,B 0.000,C 90.000,E1 200.174} C_DIS
LIN {X -0.040,Y -139.012,Z 1629.102,A 0.000,B 0.000,C 90.000,E1 198.308} C_DIS
LIN {X -0.046,Y -138.341,Z 1629.055,A 0.000,B 0.000,C 90.000,E1 189.905} C_DIS
LIN {X -0.026,Y -139.398,Z 1629.008,A 0.000,B 0.000,C 90.000,E1 181.489} C_DIS
LIN {X 0.028,Y -141.302,Z 1628.972,A 0.000,B 0.000,C 90.000,E1 174.951} C_DIS
LIN {X -0.015,Y -142.663,Z 1628.957,A 0.000,B 0.000,C 90.000,E1 172.186} C_DIS
LIN {X -0.065,Y -145.009,Z 1628.931,A 0.000,B 0.000,C 90.000,E1 167.589} C_DIS
LIN {X -0.076,Y -147.636,Z 1628.911,A 0.000,B 0.000,C 90.000,E1 163.921} C_DIS
LIN {X 0.002,Y -150.266,Z 1628.890,A 0.000,B 0.000,C 90.000,E1 160.242} C_DIS
LIN {X 0.015,Y -153.666,Z 1628.870,A 0.000,B 0.000,C 90.000,E1 156.613} C_DIS
LIN {X 0.072,Y -157.081,Z 1628.850,A 0.000,B 0.000,C 90.000,E1 152.999} C_DIS
LIN {X 0.010,Y -161.216,Z 1628.830,A 0.000,B 0.000,C 90.000,E1 149.459} C_DIS
LIN {X -0.043,Y -163.306,Z 1628.821,A 0.000,B 0.000,C 90.000,E1 147.709} C_DIS
LIN {X -0.033,Y -167.754,Z 1628.801,A 0.000,B 0.000,C 90.000,E1 144.196} C_DIS
LIN {X -0.014,Y -171.570,Z 1628.786,A 0.000,B 0.000,C 90.000,E1 141.582} C_DIS
LIN {X -0.079,Y -176.518,Z 1628.767,A 0.000,B 0.000,C 90.000,E1 138.162} C_DIS
LIN {X 0.044,Y -180.817,Z 1628.753,A 0.000,B 0.000,C 90.000,E1 135.567} C_DIS
LIN {X 0.030,Y -186.225,Z 1628.734,A 0.000,B 0.000,C 90.000,E1 132.204} C_DIS
LIN {X -0.032,Y -190.863,Z 1628.721,A 0.000,B 0.000,C 90.000,E1 129.725} C_DIS
LIN {X 0.001,Y -196.625,Z 1628.702,A 0.000,B 0.000,C 90.000,E1 126.423} C_DIS
LIN {X -0.086,Y -199.863,Z 1628.693,A 0.000,B 0.000,C 90.000,E1 124.818} C_DIS
LIN {X 0.110,Y -204.261,Z 1628.680,A 0.000,B 0.000,C 90.000,E1 122.339} C_DIS
LIN {X 0.018,Y -206.072,Z 1628.675,A 0.000,B 0.000,C 90.000,E1 121.416} C_DIS
LIN {X -0.020,Y -325.840,Z 1628.675,A 0.000,B 0.000,C 90.000,E1 121.416} C_DIS
LIN {X 0.003,Y -327.326,Z 1628.674,A 0.000,B 0.000,C 90.000,E1 121.386} C_DIS
LIN {X -0.153,Y -331.112,Z 1628.673,A 0.000,B 0.000,C 90.000,E1 121.258} C_DIS
LIN {X -0.026,Y -333.327,Z 1628.673,A 0.000,B 0.000,C 90.000,E1 121.082} C_DIS
LIN {X -0.171,Y -336.400,Z 1628.671,A 0.000,B 0.000,C 90.000,E1 120.797} C_DIS
LIN {X 0.162,Y -338.400,Z 1628.669,A 0.000,B 0.000,C 90.000,E1 120.463} C_DIS
LIN {X 0.033,Y -339.971,Z 1628.668,A 0.000,B 0.000,C 90.000,E1 120.207} C_DIS
LIN {X 0.015,Y -356.325,Z 1628.647,A 0.000,B 0.000,C 90.000,E1 116.539} C_DIS
LIN {X 0.212,Y -370.208,Z 1628.633,A 0.000,B 0.000,C 90.000,E1 113.823} C_DIS
LIN {X -0.110,Y -383.894,Z 1628.620,A 0.000,B 0.000,C 90.000,E1 111.535} C_DIS
LIN {X 0.132,Y -398.941,Z 1628.607,A 0.000,B 0.000,C 90.000,E1 109.214} C_DIS
LIN {X 0.120,Y -415.454,Z 1628.594,A 0.000,B 0.000,C 90.000,E1 106.985} C_DIS
LIN {X -0.022,Y -433.547,Z 1628.582,A 0.000,B 0.000,C 90.000,E1 104.828} C_DIS
LIN {X 0.109,Y -453.130,Z 1628.571,A 0.000,B 0.000,C 90.000,E1 102.715} C_DIS
LIN {X 0.098,Y -473.394,Z 1628.560,A 0.000,B 0.000,C 90.000,E1 100.782} C_DIS
LIN {X -0.029,Y -496.813,Z 1628.549,A 0.000,B 0.000,C 90.000,E1 98.803} C_DIS
LIN {X 0.199,Y -499.096,Z 1628.548,A 0.000,B 0.000,C 90.000,E1 98.568} C_DIS
LIN {X -0.143,Y -500.827,Z 1628.547,A 0.000,B 0.000,C 90.000,E1 98.398} C_DIS
LIN {X -0.216,Y -502.363,Z 1628.545,A 0.000,B 0.000,C 90.000,E1 98.163} C_DIS
LIN {X 0.207,Y -503.505,Z 1628.544,A 0.000,B 0.000,C 90.000,E1 97.871} C_DIS
LIN {X 0.005,Y -504.852,Z 1628.541,A 0.000,B 0.000,C 90.000,E1 97.409} C_DIS
LIN {X -0.191,Y -505.143,Z 1628.538,A 0.000,B 0.000,C 90.000,E1 96.947} C_DIS
LIN {X 0.123,Y -504.427,Z 1628.536,A 0.000,B 0.000,C 90.000,E1 96.429} C_DIS
LIN {X -0.063,Y -502.582,Z 1628.533,A 0.000,B 0.000,C 90.000,E1 95.967} C_DIS
LIN {X -0.184,Y -501.123,Z 1628.532,A 0.000,B 0.000,C 90.000,E1 95.739} C_DIS
LIN {X -0.138,Y -487.638,Z 1628.521,A 0.000,B 0.000,C 90.000,E1 93.784} C_DIS
LIN {X -0.099,Y -477.402,Z 1628.513,A 0.000,B 0.000,C 90.000,E1 92.293} C_DIS
LIN {X -0.231,Y -466.908,Z 1628.504,A 0.000,B 0.000,C 90.000,E1 90.802} C_DIS
LIN {X -0.086,Y -456.134,Z 1628.496,A 0.000,B 0.000,C 90.000,E1 89.255} C_DIS
LIN {X 0.127,Y -446.747,Z 1628.489,A 0.000,B 0.000,C 90.000,E1 87.936} C_DIS
LIN {X 0.196,Y -436.975,Z 1628.481,A 0.000,B 0.000,C 90.000,E1 86.617} C_DIS
LIN {X -0.014,Y -423.027,Z 1628.471,A 0.000,B 0.000,C 90.000,E1 84.780} C_DIS
LIN {X -0.088,Y -401.727,Z 1628.454,A 0.000,B 0.000,C 90.000,E1 81.781} C_DIS
LIN {X -0.143,Y -380.405,Z 1628.435,A 0.000,B 0.000,C 90.000,E1 78.398} C_DIS
LIN {X 0.022,Y -365.398,Z 1628.421,A 0.000,B 0.000,C 90.000,E1 75.755} C_DIS
LIN {X 0.007,Y -352.469,Z 1628.408,A 0.000,B 0.000,C 90.000,E1 73.378} C_DIS
LIN {X 0.103,Y -337.103,Z 1628.391,A 0.000,B 0.000,C 90.000,E1 70.315} C_DIS
LIN {X -0.126,Y -322.350,Z 1628.373,A 0.000,B 0.000,C 90.000,E1 67.230} C_DIS
LIN {X -0.105,Y -308.947,Z 1628.356,A 0.000,B 0.000,C 90.000,E1 64.024} C_DIS
LIN {X -0.008,Y -299.822,Z 1628.343,A 0.000,B 0.000,C 90.000,E1 61.719} C_DIS
LIN {X -0.086,Y -291.819,Z 1628.332,A 0.000,B 0.000,C 90.000,E1 59.744} C_DIS
LIN {X -0.012,Y -283.625,Z 1628.321,A 0.000,B 0.000,C 90.000,E1 57.709} C_DIS
LIN {X -0.038,Y -276.479,Z 1628.311,A 0.000,B 0.000,C 90.000,E1 56.008} C_DIS
LIN {X -0.028,Y -266.383,Z 1628.298,A 0.000,B 0.000,C 90.000,E1 53.577} C_DIS
LIN {X 0.026,Y -256.439,Z 1628.284,A 0.000,B 0.000,C 90.000,E1 51.090} C_DIS
LIN {X 0.011,Y -244.180,Z 1628.266,A 0.000,B 0.000,C 90.000,E1 47.838} C_DIS
LIN {X -0.022,Y -232.956,Z 1628.247,A 0.000,B 0.000,C 90.000,E1 44.514} C_DIS
LIN {X 0.042,Y -223.791,Z 1628.230,A 0.000,B 0.000,C 90.000,E1 41.472} C_DIS
LIN {X 0.083,Y -215.423,Z 1628.213,A 0.000,B 0.000,C 90.000,E1 38.382} C_DIS
LIN {X 0.037,Y -207.907,Z 1628.196,A 0.000,B 0.000,C 90.000,E1 35.264} C_DIS
LIN {X 0.033,Y -201.160,Z 1628.178,A 0.000,B 0.000,C 90.000,E1 32.084} C_DIS
LIN {X -0.015,Y -195.189,Z 1628.160,A 0.000,B 0.000,C 90.000,E1 28.871} C_DIS
LIN {X 0.019,Y -189.883,Z 1628.142,A 0.000,B 0.000,C 90.000,E1 25.591} C_DIS
LIN {X 0.028,Y -185.296,Z 1628.124,A 0.000,B 0.000,C 90.000,E1 22.280} C_DIS
LIN {X -0.063,Y -180.460,Z 1628.101,A 0.000,B 0.000,C 90.000,E1 18.127} C_DIS
LIN {X -0.011,Y -176.476,Z 1628.077,A 0.000,B 0.000,C 90.000,E1 13.883} C_DIS
LIN {X 0.005,Y -173.216,Z 1628.053,A 0.000,B 0.000,C 90.000,E1 9.613} C_DIS
LIN {X -0.053,Y -170.221,Z 1628.020,A 0.000,B 0.000,C 90.000,E1 3.612} C_DIS
LIN {X 0.056,Y -168.526,Z 1627.978,A 0.000,B 0.000,C 90.000,E1 356.045} C_DIS
LIN {X -0.050,Y -170.138,Z 1627.930,A 0.000,B 0.000,C 90.000,E1 347.409} C_DIS
LIN {X -0.063,Y -173.190,Z 1627.901,A 0.000,B 0.000,C 90.000,E1 342.236} C_DIS
LIN {X 0.027,Y -176.968,Z 1627.877,A 0.000,B 0.000,C 90.000,E1 337.922} C_DIS
LIN {X -0.015,Y -181.053,Z 1627.859,A 0.000,B 0.000,C 90.000,E1 334.537} C_DIS
LIN {X -0.043,Y -186.071,Z 1627.840,A 0.000,B 0.000,C 90.000,E1 331.179} C_DIS
LIN {X -0.094,Y -191.861,Z 1627.821,A 0.000,B 0.000,C 90.000,E1 327.867} C_DIS
LIN {X -0.021,Y -198.456,Z 1627.803,A 0.000,B 0.000,C 90.000,E1 324.562} C_DIS
LIN {X -0.035,Y -205.859,Z 1627.785,A 0.000,B 0.000,C 90.000,E1 321.331} C_DIS
LIN {X 0.041,Y -213.169,Z 1627.770,A 0.000,B 0.000,C 90.000,E1 318.528} C_DIS
LIN {X 0.042,Y -222.575,Z 1627.752,A 0.000,B 0.000,C 90.000,E1 315.405} C_DIS
LIN {X -0.043,Y -233.166,Z 1627.735,A 0.000,B 0.000,C 90.000,E1 312.366} C_DIS
LIN {X 0.055,Y -241.944,Z 1627.723,A 0.000,B 0.000,C 90.000,E1 310.092} C_DIS
LIN {X 0.009,Y -250.135,Z 1627.713,A 0.000,B 0.000,C 90.000,E1 308.257} C_DIS
LIN {X -0.025,Y -261.018,Z 1627.700,A 0.000,B 0.000,C 90.000,E1 306.091} C_DIS
LIN {X -0.086,Y -275.173,Z 1627.687,A 0.000,B 0.000,C 90.000,E1 303.627} C_DIS
LIN {X -0.024,Y -288.725,Z 1627.675,A 0.000,B 0.000,C 90.000,E1 301.544} C_DIS
LIN {X -0.057,Y -308.288,Z 1627.660,A 0.000,B 0.000,C 90.000,E1 298.871} C_DIS
LIN {X -0.131,Y -320.663,Z 1627.651,A 0.000,B 0.000,C 90.000,E1 297.257} C_DIS
LIN {X -0.044,Y -335.417,Z 1627.641,A 0.000,B 0.000,C 90.000,E1 295.335} C_DIS
LIN {X 0.044,Y -349.759,Z 1627.630,A 0.000,B 0.000,C 90.000,E1 293.462} C_DIS
LIN {X -0.052,Y -364.108,Z 1627.620,A 0.000,B 0.000,C 90.000,E1 291.663} C_DIS
LIN {X 0.010,Y -375.902,Z 1627.612,A 0.000,B 0.000,C 90.000,E1 290.174} C_DIS
LIN {X -0.146,Y -384.610,Z 1627.606,A 0.000,B 0.000,C 90.000,E1 289.033} C_DIS
LIN {X 0.147,Y -390.525,Z 1627.601,A 0.000,B 0.000,C 90.000,E1 288.127} C_DIS
LIN {X 0.130,Y -395.833,Z 1627.596,A 0.000,B 0.000,C 90.000,E1 287.275} C_DIS
LIN {X -0.025,Y -399.025,Z 1627.593,A 0.000,B 0.000,C 90.000,E1 286.732} C_DIS
LIN {X -0.091,Y -403.020,Z 1627.588,A 0.000,B 0.000,C 90.000,E1 285.898} C_DIS
LIN {X 0.076,Y -405.219,Z 1627.585,A 0.000,B 0.000,C 90.000,E1 285.315} C_DIS
LIN {X -0.025,Y -407.076,Z 1627.582,A 0.000,B 0.000,C 90.000,E1 284.773} C_DIS
LIN {X -0.226,Y -408.536,Z 1627.579,A 0.000,B 0.000,C 90.000,E1 284.245} C_DIS
LIN {X 0.081,Y -409.575,Z 1627.576,A 0.000,B 0.000,C 90.000,E1 283.647} C_DIS
LIN {X -0.100,Y -410.217,Z 1627.573,A 0.000,B 0.000,C 90.000,E1 283.119} C_DIS
LIN {X 0.127,Y -410.349,Z 1627.570,A 0.000,B 0.000,C 90.000,E1 282.535} C_DIS
LIN {X -0.042,Y -409.984,Z 1627.567,A 0.000,B 0.000,C 90.000,E1 282.007} C_DIS
LIN {X 0.191,Y -409.085,Z 1627.564,A 0.000,B 0.000,C 90.000,E1 281.422} C_DIS
LIN {X 0.019,Y -407.655,Z 1627.561,A 0.000,B 0.000,C 90.000,E1 280.894} C_DIS
LIN {X -0.158,Y -405.476,Z 1627.557,A 0.000,B 0.000,C 90.000,E1 280.366} C_DIS
LIN {X -0.055,Y -404.247,Z 1627.556,A 0.000,B 0.000,C 90.000,E1 280.074} C_DIS
LIN {X 0.074,Y -401.096,Z 1627.553,A 0.000,B 0.000,C 90.000,E1 279.500} C_DIS
LIN {X -0.141,Y -397.366,Z 1627.550,A 0.000,B 0.000,C 90.000,E1 278.973} C_DIS
LIN {X 0.027,Y -390.727,Z 1627.545,A 0.000,B 0.000,C 90.000,E1 278.106} C_DIS
LIN {X 0.163,Y -382.967,Z 1627.540,A 0.000,B 0.000,C 90.000,E1 277.239} C_DIS
LIN {X -0.023,Y -377.391,Z 1627.537,A 0.000,B 0.000,C 90.000,E1 276.720} C_DIS
LIN {X -0.001,Y -371.562,Z 1627.534,A 0.000,B 0.000,C 90.000,E1 276.201} C_DIS
LIN {X -0.100,Y -365.487,Z 1627.532,A 0.000,B 0.000,C 90.000,E1 275.739} C_DIS
LIN {X 0.047,Y -359.235,Z 1627.529,A 0.000,B 0.000,C 90.000,E1 275.277} C_DIS
LIN {X -0.048,Y -349.686,Z 1627.526,A 0.000,B 0.000,C 90.000,E1 274.702} C_DIS
LIN {X -0.060,Y -339.985,Z 1627.523,A 0.000,B 0.000,C 90.000,E1 274.188} C_DIS
LIN {X -0.103,Y -330.184,Z 1627.521,A 0.000,B 0.000,C 90.000,E1 273.726} C_DIS
LIN {X 0.124,Y -320.457,Z 1627.518,A 0.000,B 0.000,C 90.000,E1 273.269} C_DIS
LIN {X -0.052,Y -310.258,Z 1627.516,A 0.000,B 0.000,C 90.000,E1 272.922} C_DIS
LIN {X 0.059,Y -299.692,Z 1627.514,A 0.000,B 0.000,C 90.000,E1 272.579} C_DIS
LIN {X -0.134,Y -288.210,Z 1627.513,A 0.000,B 0.000,C 90.000,E1 272.350} C_DIS
LIN {X 0.010,Y -279.459,Z 1627.512,A 0.000,B 0.000,C 90.000,E1 272.178} C_DIS
LIN {X 0.048,Y -263.952,Z 1627.511,A 0.000,B 0.000,C 90.000,E1 272.007} C_DIS
LIN {X 0.112,Y -229.780,Z 1627.510,A 0.000,B 0.000,C 90.000,E1 271.718} C_DIS
LIN {X 0.025,Y -212.292,Z 1627.509,A 0.000,B 0.000,C 90.000,E1 271.661} C_DIS
LIN {X -0.014,Y -206.235,Z 1627.509,A 0.000,B 0.000,C 90.000,E1 271.661} C_DIS
LIN {X -0.047,Y -181.323,Z 1627.509,A 0.000,B 0.000,C 90.000,E1 271.661} C_DIS
LIN {X -0.042,Y -181.548,Z 1627.500,A 0.000,B 0.000,C 90.000,E1 269.943} C_DIS
LIN {X -0.057,Y -180.829,Z 1627.472,A 0.000,B 0.000,C 90.000,E1 264.894} C_DIS
LIN {X 0.022,Y -178.934,Z 1627.443,A 0.000,B 0.000,C 90.000,E1 259.803} C_DIS
LIN {X 0.060,Y -175.983,Z 1627.415,A 0.000,B 0.000,C 90.000,E1 254.700} C_DIS
LIN {X 0.005,Y -175.478,Z 1627.410,A 0.000,B 0.000,C 90.000,E1 253.866} C_DIS
LIN {X 0.062,Y -172.225,Z 1627.387,A 0.000,B 0.000,C 90.000,E1 249.571} C_DIS
LIN {X 0.039,Y -171.701,Z 1627.382,A 0.000,B 0.000,C 90.000,E1 248.720} C_DIS
LIN {X -0.036,Y -167.296,Z 1627.353,A 0.000,B 0.000,C 90.000,E1 243.563} C_DIS
LIN {X 0.047,Y -166.673,Z 1627.348,A 0.000,B 0.000,C 90.000,E1 242.666} C_DIS
LIN {X -0.038,Y -162.656,Z 1627.324,A 0.000,B 0.000,C 90.000,E1 238.329} C_DIS
LIN {X 0.025,Y -161.345,Z 1627.314,A 0.000,B 0.000,C 90.000,E1 236.548} C_DIS
LIN {X 0.067,Y -157.340,Z 1627.290,A 0.000,B 0.000,C 90.000,E1 232.110} C_DIS
LIN {X -0.001,Y -155.324,Z 1627.275,A 0.000,B 0.000,C 90.000,E1 229.461} C_DIS
LIN {X -0.070,Y -151.677,Z 1627.250,A 0.000,B 0.000,C 90.000,E1 225.000} C_DIS
LIN {X -0.021,Y -150.542,Z 1627.240,A 0.000,B 0.000,C 90.000,E1 223.176} C_DIS
LIN {X 0.011,Y -147.267,Z 1627.215,A 0.000,B 0.000,C 90.000,E1 218.624} C_DIS
LIN {X -0.016,Y -145.294,Z 1627.194,A 0.000,B 0.000,C 90.000,E1 214.978} C_DIS
LIN {X -0.023,Y -142.391,Z 1627.164,A 0.000,B 0.000,C 90.000,E1 209.461} C_DIS
LIN {X 0.023,Y -141.370,Z 1627.148,A 0.000,B 0.000,C 90.000,E1 206.668} C_DIS
LIN {X 0.001,Y -139.345,Z 1627.112,A 0.000,B 0.000,C 90.000,E1 200.174} C_DIS
LIN {X 0.006,Y -139.018,Z 1627.102,A 0.000,B 0.000,C 90.000,E1 198.308} C_DIS
LIN {X 0.002,Y -138.342,Z 1627.055,A 0.000,B 0.000,C 90.000,E1 189.905} C_DIS
LIN {X 0.021,Y -139.393,Z 1627.008,A 0.000,B 0.000,C 90.000,E1 181.489} C_DIS
LIN {X -0.065,Y -141.293,Z 1626.972,A 0.000,B 0.000,C 90.000,E1 175.008} C_DIS
LIN {X 0.033,Y -142.655,Z 1626.957,A 0.000,B 0.000,C 90.000,E1 172.186} C_DIS
LIN {X -0.017,Y -144.997,Z 1626.931,A 0.000,B 0.000,C 90.000,E1 167.589} C_DIS
LIN {X -0.027,Y -147.624,Z 1626.911,A 0.000,B 0.000,C 90.000,E1 163.921} C_DIS
LIN {X 0.051,Y -150.250,Z 1626.890,A 0.000,B 0.000,C 90.000,E1 160.242} C_DIS
LIN {X 0.065,Y -153.647,Z 1626.870,A 0.000,B 0.000,C 90.000,E1 156.613} C_DIS
LIN {X -0.017,Y -157.062,Z 1626.850,A 0.000,B 0.000,C 90.000,E1 153.050} C_DIS
LIN {X 0.062,Y -161.193,Z 1626.830,A 0.000,B 0.000,C 90.000,E1 149.459} C_DIS
LIN {X 0.010,Y -163.286,Z 1626.821,A 0.000,B 0.000,C 90.000,E1 147.709} C_DIS
LIN {X 0.020,Y -167.729,Z 1626.801,A 0.000,B 0.000,C 90.000,E1 144.196} C_DIS
LIN {X -0.068,Y -171.547,Z 1626.787,A 0.000,B 0.000,C 90.000,E1 141.618} C_DIS
LIN {X -0.025,Y -176.490,Z 1626.768,A 0.000,B 0.000,C 90.000,E1 138.162} C_DIS
LIN {X 0.100,Y -180.788,Z 1626.753,A 0.000,B 0.000,C 90.000,E1 135.567} C_DIS
LIN {X -0.039,Y -186.195,Z 1626.735,A 0.000,B 0.000,C 90.000,E1 132.243} C_DIS
LIN {X 0.025,Y -190.833,Z 1626.721,A 0.000,B 0.000,C 90.000,E1 129.725} C_DIS
LIN {X -0.057,Y -196.592,Z 1626.702,A 0.000,B 0.000,C 90.000,E1 126.457} C_DIS
LIN {X 0.027,Y -201.359,Z 1626.689,A 0.000,B 0.000,C 90.000,E1 123.992} C_DIS
LIN {X -0.008,Y -205.990,Z 1626.675,A 0.000,B 0.000,C 90.000,E1 121.465} C_DIS
LIN {X -0.048,Y -325.552,Z 1626.675,A 0.000,B 0.000,C 90.000,E1 121.465} C_DIS
LIN {X 0.098,Y -328.080,Z 1626.674,A 0.000,B 0.000,C 90.000,E1 121.386} C_DIS
LIN {X 0.070,Y -333.454,Z 1626.673,A 0.000,B 0.000,C 90.000,E1 121.082} C_DIS
LIN {X -0.074,Y -336.421,Z 1626.671,A 0.000,B 0.000,C 90.000,E1 120.797} C_DIS
LIN {X -0.075,Y -338.415,Z 1626.669,A 0.000,B 0.000,C 90.000,E1 120.512} C_DIS
LIN {X 0.044,Y -339.977,Z 1626.668,A 0.000,B 0.000,C 90.000,E1 120.207} C_DIS
LIN {X -0.164,Y -354.843,Z 1626.649,A 0.000,B 0.000,C 90.000,E1 116.873} C_DIS
LIN {X -0.013,Y -368.558,Z 1626.634,A 0.000,B 0.000,C 90.000,E1 114.155} C_DIS
LIN {X -0.229,Y -382.079,Z 1626.621,A 0.000,B 0.000,C 90.000,E1 111.844} C_DIS
LIN {X 0.094,Y -396.950,Z 1626.608,A 0.000,B 0.000,C 90.000,E1 109.504} C_DIS
LIN {X 0.020,Y -413.273,Z 1626.596,A 0.000,B 0.000,C 90.000,E1 107.275} C_DIS
LIN {X 0.118,Y -431.162,Z 1626.584,A 0.000,B 0.000,C 90.000,E1 105.079} C_DIS
LIN {X -0.196,Y -450.611,Z 1626.572,A 0.000,B 0.000,C 90.000,E1 103.008} C_DIS
LIN {X 0.160,Y -470.806,Z 1626.561,A 0.000,B 0.000,C 90.000,E1 101.007} C_DIS
LIN {X -0.134,Y -494.130,Z 1626.550,A 0.000,B 0.000,C 90.000,E1 99.029} C_DIS
LIN {X -0.023,Y -496.773,Z 1626.549,A 0.000,B 0.000,C 90.000,E1 98.803} C_DIS
LIN {X 0.204,Y -499.025,Z 1626.548,A 0.000,B 0.000,C 90.000,E1 98.568} C_DIS
LIN {X -0.137,Y -500.734,Z 1626.547,A 0.000,B 0.000,C 90.000,E1 98.398} C_DIS
LIN {X -0.211,Y -502.251,Z 1626.545,A 0.000,B 0.000,C 90.000,E1 98.163} C_DIS
LIN {X 0.211,Y -503.378,Z 1626.544,A 0.000,B 0.000,C 90.000,E1 97.871} C_DIS
LIN {X 0.009,Y -504.702,Z 1626.541,A 0.000,B 0.000,C 90.000,E1 97.409} C_DIS
LIN {X -0.187,Y -504.972,Z 1626.538,A 0.000,B 0.000,C 90.000,E1 96.947} C_DIS
LIN {X 0.126,Y -504.236,Z 1626.536,A 0.000,B 0.000,C 90.000,E1 96.429} C_DIS
LIN {X -0.061,Y -502.366,Z 1626.533,A 0.000,B 0.000,C 90.000,E1 95.967} C_DIS
LIN {X 0.197,Y -499.184,Z 1626.530,A 0.000,B 0.000,C 90.000,E1 95.454} C_DIS
LIN {X -0.141,Y -487.406,Z 1626.521,A 0.000,B 0.000,C 90.000,E1 93.784} C_DIS
LIN {X -0.106,Y -477.204,Z 1626.513,A 0.000,B 0.000,C 90.000,E1 92.293} C_DIS
LIN {X -0.046,Y -468.487,Z 1626.506,A 0.000,B 0.000,C 90.000,E1 91.031} C_DIS
LIN {X 0.122,Y -457.772,Z 1626.497,A 0.000,B 0.000,C 90.000,E1 89.484} C_DIS
LIN {X -0.113,Y -448.452,Z 1626.490,A 0.000,B 0.000,C 90.000,E1 88.224} C_DIS
LIN {X -0.016,Y -438.749,Z 1626.483,A 0.000,B 0.000,C 90.000,E1 86.906} C_DIS
LIN {X 0.100,Y -426.780,Z 1626.474,A 0.000,B 0.000,C 90.000,E1 85.298} C_DIS
LIN {X -0.035,Y -409.046,Z 1626.460,A 0.000,B 0.000,C 90.000,E1 82.875} C_DIS
LIN {X 0.027,Y -387.083,Z 1626.442,A 0.000,B 0.000,C 90.000,E1 79.511} C_DIS
LIN {X -0.080,Y -371.766,Z 1626.427,A 0.000,B 0.000,C 90.000,E1 76.937} C_DIS
LIN {X -0.034,Y -358.691,Z 1626.414,A 0.000,B 0.000,C 90.000,E1 74.574} C_DIS
LIN {X -0.180,Y -342.931,Z 1626.397,A 0.000,B 0.000,C 90.000,E1 71.583} C_DIS
LIN {X 0.027,Y -332.372,Z 1626.385,A 0.000,B 0.000,C 90.000,E1 69.390} C_DIS
LIN {X 0.069,Y -320.745,Z 1626.372,A 0.000,B 0.000,C 90.000,E1 66.869} C_DIS
LIN {X -0.161,Y -308.755,Z 1626.355,A 0.000,B 0.000,C 90.000,E1 64.024} C_DIS
LIN {X -0.065,Y -299.660,Z 1626.343,A 0.000,B 0.000,C 90.000,E1 61.719} C_DIS
LIN {X -0.146,Y -291.695,Z 1626.332,A 0.000,B 0.000,C 90.000,E1 59.744} C_DIS
LIN {X -0.073,Y -283.474,Z 1626.321,A 0.000,B 0.000,C 90.000,E1 57.709} C_DIS
LIN {X -0.100,Y -276.329,Z 1626.311,A 0.000,B 0.000,C 90.000,E1 56.008} C_DIS
LIN {X 0.068,Y -266.192,Z 1626.297,A 0.000,B 0.000,C 90.000,E1 53.543} C_DIS
LIN {X -0.039,Y -256.175,Z 1626.284,A 0.000,B 0.000,C 90.000,E1 51.090} C_DIS
LIN {X -0.057,Y -243.900,Z 1626.266,A 0.000,B 0.000,C 90.000,E1 47.838} C_DIS
LIN {X -0.094,Y -232.691,Z 1626.247,A 0.000,B 0.000,C 90.000,E1 44.514} C_DIS
LIN {X -0.034,Y -223.569,Z 1626.230,A 0.000,B 0.000,C 90.000,E1 41.472} C_DIS
LIN {X 0.005,Y -215.240,Z 1626.213,A 0.000,B 0.000,C 90.000,E1 38.382} C_DIS
LIN {X 0.076,Y -207.770,Z 1626.196,A 0.000,B 0.000,C 90.000,E1 35.231} C_DIS
LIN {X -0.048,Y -201.066,Z 1626.178,A 0.000,B 0.000,C 90.000,E1 32.084} C_DIS
LIN {X 0.075,Y -195.106,Z 1626.160,A 0.000,B 0.000,C 90.000,E1 28.821} C_DIS
LIN {X -0.061,Y -189.835,Z 1626.142,A 0.000,B 0.000,C 90.000,E1 25.591} C_DIS
LIN {X -0.051,Y -185.296,Z 1626.124,A 0.000,B 0.000,C 90.000,E1 22.280} C_DIS
LIN {X 0.087,Y -180.490,Z 1626.100,A 0.000,B 0.000,C 90.000,E1 18.055} C_DIS
LIN {X 0.086,Y -176.535,Z 1626.077,A 0.000,B 0.000,C 90.000,E1 13.828} C_DIS
LIN {X -0.066,Y -173.311,Z 1626.053,A 0.000,B 0.000,C 90.000,E1 9.613} C_DIS
LIN {X 0.052,Y -170.358,Z 1626.020,A 0.000,B 0.000,C 90.000,E1 3.555} C_DIS
LIN {X 0.055,Y -168.634,Z 1625.973,A 0.000,B 0.000,C 90.000,E1 355.179} C_DIS
LIN {X -0.037,Y -170.308,Z 1625.930,A 0.000,B 0.000,C 90.000,E1 347.409} C_DIS
LIN {X -0.044,Y -173.345,Z 1625.901,A 0.000,B 0.000,C 90.000,E1 342.236} C_DIS
LIN {X 0.059,Y -176.275,Z 1625.882,A 0.000,B 0.000,C 90.000,E1 338.773} C_DIS
LIN {X -0.067,Y -180.124,Z 1625.863,A 0.000,B 0.000,C 90.000,E1 335.409} C_DIS
LIN {X -0.035,Y -184.900,Z 1625.844,A 0.000,B 0.000,C 90.000,E1 332.025} C_DIS
LIN {X 0.053,Y -190.527,Z 1625.826,A 0.000,B 0.000,C 90.000,E1 328.663} C_DIS
LIN {X -0.009,Y -196.895,Z 1625.808,A 0.000,B 0.000,C 90.000,E1 325.388} C_DIS
LIN {X -0.020,Y -204.103,Z 1625.790,A 0.000,B 0.000,C 90.000,E1 322.145} C_DIS
LIN {X 0.030,Y -211.136,Z 1625.774,A 0.000,B 0.000,C 90.000,E1 319.337} C_DIS
LIN {X -0.032,Y -220.209,Z 1625.757,A 0.000,B 0.000,C 90.000,E1 316.215} C_DIS
LIN {X -0.023,Y -230.482,Z 1625.740,A 0.000,B 0.000,C 90.000,E1 313.137} C_DIS
LIN {X -0.009,Y -240.407,Z 1625.725,A 0.000,B 0.000,C 90.000,E1 310.496} C_DIS
LIN {X 0.084,Y -248.392,Z 1625.715,A 0.000,B 0.000,C 90.000,E1 308.624} C_DIS
LIN {X 0.020,Y -259.053,Z 1625.703,A 0.000,B 0.000,C 90.000,E1 306.457} C_DIS
LIN {X -0.085,Y -272.999,Z 1625.689,A 0.000,B 0.000,C 90.000,E1 303.992} C_DIS
LIN {X 0.090,Y -286.297,Z 1625.677,A 0.000,B 0.000,C 90.000,E1 301.878} C_DIS
LIN {X 0.003,Y -305.746,Z 1625.662,A 0.000,B 0.000,C 90.000,E1 299.205} C_DIS
LIN {X -0.043,Y -320.618,Z 1625.651,A 0.000,B 0.000,C 90.000,E1 297.257} C_DIS
LIN {X 0.046,Y -335.350,Z 1625.641,A 0.000,B 0.000,C 90.000,E1 295.335} C_DIS
LIN {X -0.183,Y -349.674,Z 1625.630,A 0.000,B 0.000,C 90.000,E1 293.515} C_DIS
LIN {X -0.011,Y -361.638,Z 1625.622,A 0.000,B 0.000,C 90.000,E1 291.972} C_DIS
LIN {X 0.008,Y -373.557,Z 1625.614,A 0.000,B 0.000,C 90.000,E1 290.482} C_DIS
LIN {X -0.162,Y -380.317,Z 1625.609,A 0.000,B 0.000,C 90.000,E1 289.631} C_DIS
LIN {X 0.084,Y -386.621,Z 1625.604,A 0.000,B 0.000,C 90.000,E1 288.725} C_DIS
LIN {X 0.031,Y -392.384,Z 1625.599,A 0.000,B 0.000,C 90.000,E1 287.873} C_DIS
LIN {X -0.096,Y -397.528,Z 1625.595,A 0.000,B 0.000,C 90.000,E1 287.040} C_DIS
LIN {X -0.171,Y -401.882,Z 1625.590,A 0.000,B 0.000,C 90.000,E1 286.205} C_DIS
LIN {X -0.208,Y -405.359,Z 1625.585,A 0.000,B 0.000,C 90.000,E1 285.371} C_DIS
LIN {X 0.082,Y -407.232,Z 1625.582,A 0.000,B 0.000,C 90.000,E1 284.773} C_DIS
LIN {X -0.117,Y -408.739,Z 1625.579,A 0.000,B 0.000,C 90.000,E1 284.245} C_DIS
LIN {X 0.191,Y -409.832,Z 1625.576,A 0.000,B 0.000,C 90.000,E1 283.647} C_DIS
LIN {X 0.012,Y -410.505,Z 1625.573,A 0.000,B 0.000,C 90.000,E1 283.119} C_DIS
LIN {X -0.160,Y -410.633,Z 1625.570,A 0.000,B 0.000,C 90.000,E1 282.591} C_DIS
LIN {X 0.073,Y -410.340,Z 1625.567,A 0.000,B 0.000,C 90.000,E1 282.007} C_DIS
LIN {X -0.094,Y -409.489,Z 1625.564,A 0.000,B 0.000,C 90.000,E1 281.478} C_DIS
LIN {X 0.137,Y -408.064,Z 1625.561,A 0.000,B 0.000,C 90.000,E1 280.894} C_DIS
LIN {X -0.038,Y -406.017,Z 1625.558,A 0.000,B 0.000,C 90.000,E1 280.366} C_DIS
LIN {X 0.106,Y -403.289,Z 1625.554,A 0.000,B 0.000,C 90.000,E1 279.792} C_DIS
LIN {X -0.097,Y -399.878,Z 1625.551,A 0.000,B 0.000,C 90.000,E1 279.265} C_DIS
LIN {X 0.074,Y -395.887,Z 1625.548,A 0.000,B 0.000,C 90.000,E1 278.681} C_DIS
LIN {X 0.160,Y -391.376,Z 1625.545,A 0.000,B 0.000,C 90.000,E1 278.106} C_DIS
LIN {X -0.105,Y -383.584,Z 1625.540,A 0.000,B 0.000,C 90.000,E1 277.296} C_DIS
LIN {X 0.083,Y -377.969,Z 1625.537,A 0.000,B 0.000,C 90.000,E1 276.720} C_DIS
LIN {X 0.139,Y -372.143,Z 1625.535,A 0.000,B 0.000,C 90.000,E1 276.201} C_DIS
LIN {X 0.046,Y -366.101,Z 1625.532,A 0.000,B 0.000,C 90.000,E1 275.739} C_DIS
LIN {X -0.162,Y -359.841,Z 1625.530,A 0.000,B 0.000,C 90.000,E1 275.334} C_DIS
LIN {X 0.145,Y -350.381,Z 1625.526,A 0.000,B 0.000,C 90.000,E1 274.702} C_DIS
LIN {X 0.121,Y -340.726,Z 1625.523,A 0.000,B 0.000,C 90.000,E1 274.188} C_DIS
LIN {X 0.111,Y -331.072,Z 1625.521,A 0.000,B 0.000,C 90.000,E1 273.726} C_DIS
LIN {X -0.009,Y -321.196,Z 1625.518,A 0.000,B 0.000,C 90.000,E1 273.326} C_DIS
LIN {X 0.135,Y -310.998,Z 1625.516,A 0.000,B 0.000,C 90.000,E1 272.922} C_DIS
LIN {X -0.143,Y -304.187,Z 1625.515,A 0.000,B 0.000,C 90.000,E1 272.751} C_DIS
LIN {X -0.133,Y -293.355,Z 1625.514,A 0.000,B 0.000,C 90.000,E1 272.465} C_DIS
LIN {X -0.065,Y -285.419,Z 1625.513,A 0.000,B 0.000,C 90.000,E1 272.293} C_DIS
LIN {X 0.122,Y -276.121,Z 1625.512,A 0.000,B 0.000,C 90.000,E1 272.121} C_DIS
LIN {X -0.080,Y -259.623,Z 1625.511,A 0.000,B 0.000,C 90.000,E1 272.007} C_DIS
LIN {X -0.038,Y -231.343,Z 1625.510,A 0.000,B 0.000,C 90.000,E1 271.776} C_DIS
LIN {X 0.099,Y -215.869,Z 1625.509,A 0.000,B 0.000,C 90.000,E1 271.661} C_DIS
LIN {X 0.056,Y -209.659,Z 1625.509,A 0.000,B 0.000,C 90.000,E1 271.661} C_DIS
LIN {X 0.013,Y -181.320,Z 1625.509,A 0.000,B 0.000,C 90.000,E1 271.661} C_DIS
LIN {X 0.016,Y -181.552,Z 1625.500,A 0.000,B 0.000,C 90.000,E1 269.943} C_DIS
LIN {X 0.001,Y -180.835,Z 1625.472,A 0.000,B 0.000,C 90.000,E1 264.894} C_DIS
LIN {X 0.080,Y -178.941,Z 1625.443,A 0.000,B 0.000,C 90.000,E1 259.803} C_DIS
LIN {X -0.052,Y -175.992,Z 1625.415,A 0.000,B 0.000,C 90.000,E1 254.755} C_DIS
LIN {X 0.062,Y -175.494,Z 1625.411,A 0.000,B 0.000,C 90.000,E1 253.866} C_DIS
LIN {X -0.044,Y -172.236,Z 1625.387,A 0.000,B 0.000,C 90.000,E1 249.625} C_DIS
LIN {X -0.064,Y -171.714,Z 1625.382,A 0.000,B 0.000,C 90.000,E1 248.773} C_DIS
LIN {X 0.020,Y -167.309,Z 1625.353,A 0.000,B 0.000,C 90.000,E1 243.563} C_DIS
LIN {X 0.026,Y -166.690,Z 1625.348,A 0.000,B 0.000,C 90.000,E1 242.692} C_DIS
LIN {X 0.017,Y -162.671,Z 1625.324,A 0.000,B 0.000,C 90.000,E1 238.329} C_DIS
LIN {X -0.011,Y -161.361,Z 1625.314,A 0.000,B 0.000,C 90.000,E1 236.580} C_DIS
LIN {X 0.024,Y -157.355,Z 1625.290,A 0.000,B 0.000,C 90.000,E1 232.145} C_DIS
LIN {X 0.053,Y -155.343,Z 1625.275,A 0.000,B 0.000,C 90.000,E1 229.461} C_DIS
LIN {X -0.018,Y -151.691,Z 1625.250,A 0.000,B 0.000,C 90.000,E1 225.000} C_DIS
LIN {X 0.030,Y -150.553,Z 1625.240,A 0.000,B 0.000,C 90.000,E1 223.176} C_DIS
LIN {X -0.052,Y -147.279,Z 1625.215,A 0.000,B 0.000,C 90.000,E1 218.669} C_DIS
LIN {X 0.035,Y -145.308,Z 1625.194,A 0.000,B 0.000,C 90.000,E1 214.978} C_DIS
LIN {X 0.027,Y -142.398,Z 1625.164,A 0.000,B 0.000,C 90.000,E1 209.461} C_DIS
LIN {X 0.009,Y -141.380,Z 1625.148,A 0.000,B 0.000,C 90.000,E1 206.693} C_DIS
LIN {X 0.050,Y -139.348,Z 1625.112,A 0.000,B 0.000,C 90.000,E1 200.174} C_DIS
LIN {X -0.008,Y -138.786,Z 1625.097,A 0.000,B 0.000,C 90.000,E1 197.402} C_DIS
LIN {X 0.051,Y -138.344,Z 1625.055,A 0.000,B 0.000,C 90.000,E1 189.905} C_DIS
LIN {X 0.071,Y -139.387,Z 1625.008,A 0.000,B 0.000,C 90.000,E1 181.489} C_DIS
LIN {X -0.016,Y -141.283,Z 1624.972,A 0.000,B 0.000,C 90.000,E1 175.008} C_DIS
LIN {X -0.058,Y -142.647,Z 1624.957,A 0.000,B 0.000,C 90.000,E1 172.243} C_DIS
LIN {X 0.035,Y -144.984,Z 1624.931,A 0.000,B 0.000,C 90.000,E1 167.589} C_DIS
LIN {X 0.024,Y -147.611,Z 1624.911,A 0.000,B 0.000,C 90.000,E1 163.921} C_DIS
LIN {X -0.038,Y -150.234,Z 1624.891,A 0.000,B 0.000,C 90.000,E1 160.296} C_DIS
LIN {X -0.023,Y -153.626,Z 1624.870,A 0.000,B 0.000,C 90.000,E1 156.666} C_DIS
LIN {X -0.035,Y -157.041,Z 1624.850,A 0.000,B 0.000,C 90.000,E1 153.076} C_DIS
LIN {X 0.035,Y -161.167,Z 1624.831,A 0.000,B 0.000,C 90.000,E1 149.488} C_DIS
LIN {X -0.022,Y -163.262,Z 1624.821,A 0.000,B 0.000,C 90.000,E1 147.740} C_DIS
LIN {X 0.076,Y -167.703,Z 1624.801,A 0.000,B 0.000,C 90.000,E1 144.196} C_DIS
LIN {X -0.011,Y -171.522,Z 1624.787,A 0.000,B 0.000,C 90.000,E1 141.618} C_DIS
LIN {X 0.032,Y -176.462,Z 1624.768,A 0.000,B 0.000,C 90.000,E1 138.162} C_DIS
LIN {X -0.097,Y -180.758,Z 1624.753,A 0.000,B 0.000,C 90.000,E1 135.648} C_DIS
LIN {X 0.021,Y -186.163,Z 1624.735,A 0.000,B 0.000,C 90.000,E1 132.243} C_DIS
LIN {X 0.085,Y -190.801,Z 1624.721,A 0.000,B 0.000,C 90.000,E1 129.725} C_DIS
LIN {X 0.004,Y -196.557,Z 1624.703,A 0.000,B 0.000,C 90.000,E1 126.457} C_DIS
LIN {X 0.089,Y -201.329,Z 1624.689,A 0.000,B 0.000,C 90.000,E1 123.992} C_DIS
LIN {X -0.026,Y -205.904,Z 1624.675,A 0.000,B 0.000,C 90.000,E1 121.514} C_DIS
LIN {X 0.187,Y -325.113,Z 1624.675,A 0.000,B 0.000,C 90.000,E1 121.465} C_DIS
LIN {X 0.088,Y -326.437,Z 1624.675,A 0.000,B 0.000,C 90.000,E1 121.465} C_DIS
LIN {X -0.154,Y -330.816,Z 1624.674,A 0.000,B 0.000,C 90.000,E1 121.337} C_DIS
LIN {X 0.059,Y -333.189,Z 1624.673,A 0.000,B 0.000,C 90.000,E1 121.131} C_DIS
LIN {X 0.029,Y -336.422,Z 1624.671,A 0.000,B 0.000,C 90.000,E1 120.797} C_DIS
LIN {X -0.152,Y -338.381,Z 1624.670,A 0.000,B 0.000,C 90.000,E1 120.541} C_DIS
LIN {X 0.133,Y -339.917,Z 1624.668,A 0.000,B 0.000,C 90.000,E1 120.207} C_DIS
LIN {X -0.075,Y -354.752,Z 1624.649,A 0.000,B 0.000,C 90.000,E1 116.873} C_DIS
LIN {X 0.077,Y -368.459,Z 1624.634,A 0.000,B 0.000,C 90.000,E1 114.155} C_DIS
LIN {X -0.139,Y -381.972,Z 1624.621,A 0.000,B 0.000,C 90.000,E1 111.844} C_DIS
LIN {X 0.053,Y -396.834,Z 1624.609,A 0.000,B 0.000,C 90.000,E1 109.523} C_DIS
LIN {X 0.112,Y -413.148,Z 1624.596,A 0.000,B 0.000,C 90.000,E1 107.275} C_DIS
LIN {X -0.205,Y -431.026,Z 1624.584,A 0.000,B 0.000,C 90.000,E1 105.134} C_DIS
LIN {X -0.105,Y -450.469,Z 1624.572,A 0.000,B 0.000,C 90.000,E1 103.008} C_DIS
LIN {X 0.247,Y -470.661,Z 1624.561,A 0.000,B 0.000,C 90.000,E1 101.007} C_DIS
LIN {X -0.052,Y -493.982,Z 1624.550,A 0.000,B 0.000,C 90.000,E1 99.029} C_DIS
LIN {X 0.059,Y -496.625,Z 1624.549,A 0.000,B 0.000,C 90.000,E1 98.803} C_DIS
LIN {X -0.208,Y -498.875,Z 1624.548,A 0.000,B 0.000,C 90.000,E1 98.624} C_DIS
LIN {X -0.057,Y -500.581,Z 1624.547,A 0.000,B 0.000,C 90.000,E1 98.398} C_DIS
LIN {X -0.130,Y -502.095,Z 1624.545,A 0.000,B 0.000,C 90.000,E1 98.163} C_DIS
LIN {X -0.276,Y -503.221,Z 1624.544,A 0.000,B 0.000,C 90.000,E1 97.936} C_DIS
LIN {X 0.089,Y -504.540,Z 1624.541,A 0.000,B 0.000,C 90.000,E1 97.409} C_DIS
LIN {X -0.108,Y -504.807,Z 1624.539,A 0.000,B 0.000,C 90.000,E1 96.947} C_DIS
LIN {X 0.203,Y -504.067,Z 1624.536,A 0.000,B 0.000,C 90.000,E1 96.429} C_DIS
LIN {X 0.015,Y -502.194,Z 1624.533,A 0.000,B 0.000,C 90.000,E1 95.967} C_DIS
LIN {X -0.225,Y -499.013,Z 1624.531,A 0.000,B 0.000,C 90.000,E1 95.511} C_DIS
LIN {X -0.072,Y -487.233,Z 1624.521,A 0.000,B 0.000,C 90.000,E1 93.784} C_DIS
LIN {X -0.040,Y -477.081,Z 1624.513,A 0.000,B 0.000,C 90.000,E1 92.293} C_DIS
LIN {X -0.179,Y -466.602,Z 1624.504,A 0.000,B 0.000,C 90.000,E1 90.802} C_DIS
LIN {X -0.041,Y -455.838,Z 1624.496,A 0.000,B 0.000,C 90.000,E1 89.255} C_DIS
LIN {X 0.166,Y -446.407,Z 1624.489,A 0.000,B 0.000,C 90.000,E1 87.936} C_DIS
LIN {X -0.206,Y -436.611,Z 1624.481,A 0.000,B 0.000,C 90.000,E1 86.674} C_DIS
LIN {X 0.011,Y -422.646,Z 1624.471,A 0.000,B 0.000,C 90.000,E1 84.780} C_DIS
LIN {X -0.074,Y -401.357,Z 1624.454,A 0.000,B 0.000,C 90.000,E1 81.781} C_DIS
LIN {X -0.144,Y -380.035,Z 1624.435,A 0.000,B 0.000,C 90.000,E1 78.398} C_DIS
LIN {X 0.012,Y -365.044,Z 1624.421,A 0.000,B 0.000,C 90.000,E1 75.755} C_DIS
LIN {X -0.011,Y -352.113,Z 1624.408,A 0.000,B 0.000,C 90.000,E1 73.378} C_DIS
LIN {X 0.074,Y -336.735,Z 1624.391,A 0.000,B 0.000,C 90.000,E1 70.315} C_DIS
LIN {X -0.164,Y -321.986,Z 1624.373,A 0.000,B 0.000,C 90.000,E1 67.230} C_DIS
LIN {X -0.153,Y -308.603,Z 1624.356,A 0.000,B 0.000,C 90.000,E1 64.024} C_DIS
LIN {X -0.061,Y -299.537,Z 1624.343,A 0.000,B 0.000,C 90.000,E1 61.719} C_DIS
LIN {X -0.143,Y -291.611,Z 1624.332,A 0.000,B 0.000,C 90.000,E1 59.744} C_DIS
LIN {X -0.072,Y -283.373,Z 1624.321,A 0.000,B 0.000,C 90.000,E1 57.709} C_DIS
LIN {X -0.100,Y -276.208,Z 1624.311,A 0.000,B 0.000,C 90.000,E1 56.008} C_DIS
LIN {X 0.065,Y -266.032,Z 1624.297,A 0.000,B 0.000,C 90.000,E1 53.543} C_DIS
LIN {X -0.093,Y -257.410,Z 1624.286,A 0.000,B 0.000,C 90.000,E1 51.457} C_DIS
LIN {X -0.060,Y -246.287,Z 1624.270,A 0.000,B 0.000,C 90.000,E1 48.566} C_DIS
LIN {X -0.038,Y -234.887,Z 1624.251,A 0.000,B 0.000,C 90.000,E1 45.243} C_DIS
LIN {X 0.001,Y -224.485,Z 1624.232,A 0.000,B 0.000,C 90.000,E1 41.838} C_DIS
LIN {X -0.021,Y -215.101,Z 1624.213,A 0.000,B 0.000,C 90.000,E1 38.382} C_DIS
LIN {X 0.048,Y -207.679,Z 1624.196,A 0.000,B 0.000,C 90.000,E1 35.231} C_DIS
LIN {X -0.077,Y -201.004,Z 1624.178,A 0.000,B 0.000,C 90.000,E1 32.084} C_DIS
LIN {X 0.045,Y -195.061,Z 1624.160,A 0.000,B 0.000,C 90.000,E1 28.821} C_DIS
LIN {X -0.092,Y -189.817,Z 1624.142,A 0.000,B 0.000,C 90.000,E1 25.591} C_DIS
LIN {X -0.011,Y -185.312,Z 1624.124,A 0.000,B 0.000,C 90.000,E1 22.259} C_DIS
LIN {X 0.059,Y -180.548,Z 1624.100,A 0.000,B 0.000,C 90.000,E1 18.055} C_DIS
LIN {X 0.060,Y -176.619,Z 1624.077,A 0.000,B 0.000,C 90.000,E1 13.828} C_DIS
LIN {X 0.082,Y -173.416,Z 1624.053,A 0.000,B 0.000,C 90.000,E1 9.557} C_DIS
LIN {X 0.035,Y -170.511,Z 1624.020,A 0.000,B 0.000,C 90.000,E1 3.555} C_DIS
LIN {X 0.021,Y -169.103,Z 1623.954,A 0.000,B 0.000,C 90.000,E1 351.724} C_DIS
LIN {X -0.080,Y -171.353,Z 1623.920,A 0.000,B 0.000,C 90.000,E1 345.700} C_DIS
LIN {X -0.101,Y -174.159,Z 1623.896,A 0.000,B 0.000,C 90.000,E1 341.402} C_DIS
LIN {X -0.087,Y -177.325,Z 1623.877,A 0.000,B 0.000,C 90.000,E1 337.975} C_DIS
LIN {X 0.046,Y -181.403,Z 1623.859,A 0.000,B 0.000,C 90.000,E1 334.537} C_DIS
LIN {X 0.028,Y -186.415,Z 1623.840,A 0.000,B 0.000,C 90.000,E1 331.179} C_DIS
LIN {X -0.012,Y -192.226,Z 1623.821,A 0.000,B 0.000,C 90.000,E1 327.867} C_DIS
LIN {X 0.073,Y -198.784,Z 1623.803,A 0.000,B 0.000,C 90.000,E1 324.562} C_DIS
LIN {X 0.071,Y -206.162,Z 1623.785,A 0.000,B 0.000,C 90.000,E1 321.331} C_DIS
LIN {X 0.016,Y -213.441,Z 1623.770,A 0.000,B 0.000,C 90.000,E1 318.566} C_DIS
LIN {X 0.013,Y -222.776,Z 1623.752,A 0.000,B 0.000,C 90.000,E1 315.445} C_DIS
LIN {X 0.095,Y -233.240,Z 1623.735,A 0.000,B 0.000,C 90.000,E1 312.366} C_DIS
LIN {X -0.119,Y -240.406,Z 1623.725,A 0.000,B 0.000,C 90.000,E1 310.539} C_DIS
LIN {X -0.035,Y -248.363,Z 1623.715,A 0.000,B 0.000,C 90.000,E1 308.669} C_DIS
LIN {X -0.110,Y -258.988,Z 1623.703,A 0.000,B 0.000,C 90.000,E1 306.503} C_DIS
LIN {X -0.005,Y -272.918,Z 1623.689,A 0.000,B 0.000,C 90.000,E1 303.992} C_DIS
LIN {X -0.070,Y -286.221,Z 1623.677,A 0.000,B 0.000,C 90.000,E1 301.926} C_DIS
LIN {X 0.088,Y -305.668,Z 1623.662,A 0.000,B 0.000,C 90.000,E1 299.205} C_DIS
LIN {X 0.046,Y -320.539,Z 1623.651,A 0.000,B 0.000,C 90.000,E1 297.257} C_DIS
LIN {X 0.034,Y -332.835,Z 1623.643,A 0.000,B 0.000,C 90.000,E1 295.668} C_DIS
LIN {X -0.100,Y -344.807,Z 1623.634,A 0.000,B 0.000,C 90.000,E1 294.131} C_DIS
LIN {X 0.030,Y -359.198,Z 1623.624,A 0.000,B 0.000,C 90.000,E1 292.280} C_DIS
LIN {X 0.105,Y -373.523,Z 1623.614,A 0.000,B 0.000,C 90.000,E1 290.482} C_DIS
LIN {X 0.050,Y -382.476,Z 1623.607,A 0.000,B 0.000,C 90.000,E1 289.322} C_DIS
LIN {X -0.042,Y -388.604,Z 1623.603,A 0.000,B 0.000,C 90.000,E1 288.471} C_DIS
LIN {X 0.168,Y -394.208,Z 1623.598,A 0.000,B 0.000,C 90.000,E1 287.583} C_DIS
LIN {X 0.183,Y -399.145,Z 1623.593,A 0.000,B 0.000,C 90.000,E1 286.732} C_DIS
LIN {X 0.119,Y -403.234,Z 1623.588,A 0.000,B 0.000,C 90.000,E1 285.898} C_DIS
LIN {X -0.103,Y -405.509,Z 1623.585,A 0.000,B 0.000,C 90.000,E1 285.371} C_DIS
LIN {X 0.190,Y -407.440,Z 1623.582,A 0.000,B 0.000,C 90.000,E1 284.773} C_DIS
LIN {X -0.009,Y -408.943,Z 1623.579,A 0.000,B 0.000,C 90.000,E1 284.245} C_DIS
LIN {X -0.097,Y -410.095,Z 1623.576,A 0.000,B 0.000,C 90.000,E1 283.703} C_DIS
LIN {X 0.123,Y -410.770,Z 1623.573,A 0.000,B 0.000,C 90.000,E1 283.119} C_DIS
LIN {X -0.048,Y -410.977,Z 1623.570,A 0.000,B 0.000,C 90.000,E1 282.591} C_DIS
LIN {X 0.188,Y -410.710,Z 1623.567,A 0.000,B 0.000,C 90.000,E1 282.007} C_DIS
LIN {X 0.022,Y -409.847,Z 1623.564,A 0.000,B 0.000,C 90.000,E1 281.478} C_DIS
LIN {X -0.145,Y -408.464,Z 1623.561,A 0.000,B 0.000,C 90.000,E1 280.950} C_DIS
LIN {X 0.081,Y -406.485,Z 1623.558,A 0.000,B 0.000,C 90.000,E1 280.366} C_DIS
LIN {X -0.171,Y -403.795,Z 1623.555,A 0.000,B 0.000,C 90.000,E1 279.849} C_DIS
LIN {X 0.026,Y -400.455,Z 1623.552,A 0.000,B 0.000,C 90.000,E1 279.265} C_DIS
LIN {X 0.139,Y -396.492,Z 1623.548,A 0.000,B 0.000,C 90.000,E1 278.690} C_DIS
LIN {X -0.101,Y -392.006,Z 1623.545,A 0.000,B 0.000,C 90.000,E1 278.163} C_DIS
LIN {X -0.032,Y -386.944,Z 1623.542,A 0.000,B 0.000,C 90.000,E1 277.587} C_DIS
LIN {X 0.087,Y -381.400,Z 1623.539,A 0.000,B 0.000,C 90.000,E1 277.004} C_DIS
LIN {X -0.023,Y -375.548,Z 1623.536,A 0.000,B 0.000,C 90.000,E1 276.486} C_DIS
LIN {X 0.165,Y -369.649,Z 1623.533,A 0.000,B 0.000,C 90.000,E1 275.967} C_DIS
LIN {X 0.147,Y -363.389,Z 1623.531,A 0.000,B 0.000,C 90.000,E1 275.511} C_DIS
LIN {X 0.100,Y -357.164,Z 1623.528,A 0.000,B 0.000,C 90.000,E1 275.106} C_DIS
LIN {X -0.154,Y -347.591,Z 1623.525,A 0.000,B 0.000,C 90.000,E1 274.588} C_DIS
LIN {X -0.117,Y -337.751,Z 1623.522,A 0.000,B 0.000,C 90.000,E1 274.073} C_DIS
LIN {X -0.029,Y -327.896,Z 1623.520,A 0.000,B 0.000,C 90.000,E1 273.612} C_DIS
LIN {X -0.077,Y -317.802,Z 1623.518,A 0.000,B 0.000,C 90.000,E1 273.212} C_DIS
LIN {X -0.114,Y -307.857,Z 1623.516,A 0.000,B 0.000,C 90.000,E1 272.865} C_DIS
LIN {X 0.072,Y -297.110,Z 1623.514,A 0.000,B 0.000,C 90.000,E1 272.522} C_DIS
LIN {X 0.077,Y -289.677,Z 1623.513,A 0.000,B 0.000,C 90.000,E1 272.350} C_DIS
LIN {X -0.091,Y -276.726,Z 1623.512,A 0.000,B 0.000,C 90.000,E1 272.178} C_DIS
LIN {X 0.032,Y -255.112,Z 1623.511,A 0.000,B 0.000,C 90.000,E1 271.949} C_DIS
LIN {X -0.086,Y -228.484,Z 1623.510,A 0.000,B 0.000,C 90.000,E1 271.776} C_DIS
LIN {X -0.074,Y -215.279,Z 1623.509,A 0.000,B 0.000,C 90.000,E1 271.718} C_DIS
LIN {X 0.096,Y -207.548,Z 1623.509,A 0.000,B 0.000,C 90.000,E1 271.661} C_DIS
LIN {X 0.048,Y -181.318,Z 1623.509,A 0.000,B 0.000,C 90.000,E1 271.661} C_DIS
LIN {X 0.053,Y -181.554,Z 1623.500,A 0.000,B 0.000,C 90.000,E1 269.943} C_DIS
LIN {X 0.037,Y -180.837,Z 1623.472,A 0.000,B 0.000,C 90.000,E1 264.894} C_DIS
LIN {X -0.060,Y -178.945,Z 1623.444,A 0.000,B 0.000,C 90.000,E1 259.859} C_DIS
LIN {X 0.037,Y -176.399,Z 1623.420,A 0.000,B 0.000,C 90.000,E1 255.589} C_DIS
LIN {X -0.070,Y -175.503,Z 1623.411,A 0.000,B 0.000,C 90.000,E1 253.921} C_DIS
LIN {X -0.008,Y -172.244,Z 1623.387,A 0.000,B 0.000,C 90.000,E1 249.625} C_DIS
LIN {X -0.029,Y -171.722,Z 1623.382,A 0.000,B 0.000,C 90.000,E1 248.773} C_DIS
LIN {X -0.020,Y -167.318,Z 1623.353,A 0.000,B 0.000,C 90.000,E1 243.589} C_DIS
LIN {X -0.087,Y -166.700,Z 1623.348,A 0.000,B 0.000,C 90.000,E1 242.743} C_DIS
LIN {X 0.051,Y -162.680,Z 1623.324,A 0.000,B 0.000,C 90.000,E1 238.329} C_DIS
LIN {X 0.024,Y -161.371,Z 1623.314,A 0.000,B 0.000,C 90.000,E1 236.580} C_DIS
LIN {X -0.066,Y -157.364,Z 1623.290,A 0.000,B 0.000,C 90.000,E1 232.190} C_DIS
LIN {X 0.086,Y -155.354,Z 1623.275,A 0.000,B 0.000,C 90.000,E1 229.461} C_DIS
LIN {X 0.015,Y -151.699,Z 1623.250,A 0.000,B 0.000,C 90.000,E1 225.000} C_DIS
LIN {X -0.047,Y -150.560,Z 1623.240,A 0.000,B 0.000,C 90.000,E1 223.218} C_DIS
LIN {X -0.021,Y -147.287,Z 1623.215,A 0.000,B 0.000,C 90.000,E1 218.669} C_DIS
LIN {X -0.052,Y -145.316,Z 1623.194,A 0.000,B 0.000,C 90.000,E1 215.025} C_DIS
LIN {X -0.012,Y -142.403,Z 1623.164,A 0.000,B 0.000,C 90.000,E1 209.489} C_DIS
LIN {X 0.041,Y -141.387,Z 1623.148,A 0.000,B 0.000,C 90.000,E1 206.693} C_DIS
LIN {X 0.033,Y -139.350,Z 1623.112,A 0.000,B 0.000,C 90.000,E1 200.194} C_DIS
LIN {X 0.023,Y -138.788,Z 1623.097,A 0.000,B 0.000,C 90.000,E1 197.402} C_DIS
LIN {X -0.055,Y -138.345,Z 1623.055,A 0.000,B 0.000,C 90.000,E1 189.962} C_DIS
LIN {X -0.037,Y -139.384,Z 1623.009,A 0.000,B 0.000,C 90.000,E1 181.547} C_DIS
LIN {X 0.016,Y -141.278,Z 1622.972,A 0.000,B 0.000,C 90.000,E1 175.008} C_DIS
LIN {X -0.026,Y -142.643,Z 1622.957,A 0.000,B 0.000,C 90.000,E1 172.243} C_DIS
LIN {X -0.076,Y -144.976,Z 1622.931,A 0.000,B 0.000,C 90.000,E1 167.645} C_DIS
LIN {X 0.056,Y -147.604,Z 1622.911,A 0.000,B 0.000,C 90.000,E1 163.921} C_DIS
LIN {X -0.006,Y -150.224,Z 1622.891,A 0.000,B 0.000,C 90.000,E1 160.296} C_DIS
LIN {X 0.010,Y -153.613,Z 1622.870,A 0.000,B 0.000,C 90.000,E1 156.666} C_DIS
LIN {X -0.002,Y -157.029,Z 1622.850,A 0.000,B 0.000,C 90.000,E1 153.076} C_DIS
LIN {X -0.070,Y -161.152,Z 1622.831,A 0.000,B 0.000,C 90.000,E1 149.537} C_DIS
LIN {X 0.012,Y -163.249,Z 1622.821,A 0.000,B 0.000,C 90.000,E1 147.740} C_DIS
LIN {X -0.025,Y -167.686,Z 1622.801,A 0.000,B 0.000,C 90.000,E1 144.242} C_DIS
LIN {X 0.025,Y -171.507,Z 1622.787,A 0.000,B 0.000,C 90.000,E1 141.618} C_DIS
LIN {X 0.069,Y -176.442,Z 1622.768,A 0.000,B 0.000,C 90.000,E1 138.162} C_DIS
LIN {X -0.061,Y -180.739,Z 1622.754,A 0.000,B 0.000,C 90.000,E1 135.648} C_DIS
LIN {X -0.080,Y -186.144,Z 1622.735,A 0.000,B 0.000,C 90.000,E1 132.285} C_DIS
LIN {X -0.024,Y -190.781,Z 1622.721,A 0.000,B 0.000,C 90.000,E1 129.769} C_DIS
LIN {X 0.043,Y -196.537,Z 1622.703,A 0.000,B 0.000,C 90.000,E1 126.457} C_DIS
LIN {X -0.039,Y -201.309,Z 1622.689,A 0.000,B 0.000,C 90.000,E1 124.040} C_DIS
LIN {X 0.006,Y -205.829,Z 1622.675,A 0.000,B 0.000,C 90.000,E1 121.544} C_DIS
LIN {X -0.027,Y -324.765,Z 1622.675,A 0.000,B 0.000,C 90.000,E1 121.544} C_DIS
LIN {X 0.150,Y -327.442,Z 1622.675,A 0.000,B 0.000,C 90.000,E1 121.465} C_DIS
LIN {X -0.091,Y -331.098,Z 1622.674,A 0.000,B 0.000,C 90.000,E1 121.337} C_DIS
LIN {X 0.122,Y -333.337,Z 1622.673,A 0.000,B 0.000,C 90.000,E1 121.131} C_DIS
LIN {X 0.093,Y -336.457,Z 1622.671,A 0.000,B 0.000,C 90.000,E1 120.797} C_DIS
LIN {X -0.130,Y -338.412,Z 1622.670,A 0.000,B 0.000,C 90.000,E1 120.541} C_DIS
LIN {X 0.110,Y -339.938,Z 1622.668,A 0.000,B 0.000,C 90.000,E1 120.207} C_DIS
LIN {X 0.187,Y -353.319,Z 1622.651,A 0.000,B 0.000,C 90.000,E1 117.129} C_DIS
LIN {X -0.022,Y -366.855,Z 1622.636,A 0.000,B 0.000,C 90.000,E1 114.463} C_DIS
LIN {X 0.069,Y -380.207,Z 1622.623,A 0.000,B 0.000,C 90.000,E1 112.099} C_DIS
LIN {X -0.008,Y -394.897,Z 1622.610,A 0.000,B 0.000,C 90.000,E1 109.812} C_DIS
LIN {X -0.133,Y -411.026,Z 1622.598,A 0.000,B 0.000,C 90.000,E1 107.583} C_DIS
LIN {X 0.022,Y -428.704,Z 1622.585,A 0.000,B 0.000,C 90.000,E1 105.371} C_DIS
LIN {X 0.036,Y -447.980,Z 1622.574,A 0.000,B 0.000,C 90.000,E1 103.244} C_DIS
LIN {X 0.227,Y -468.103,Z 1622.563,A 0.000,B 0.000,C 90.000,E1 101.243} C_DIS
LIN {X 0.218,Y -491.383,Z 1622.551,A 0.000,B 0.000,C 90.000,E1 99.208} C_DIS
LIN {X 0.030,Y -496.634,Z 1622.549,A 0.000,B 0.000,C 90.000,E1 98.803} C_DIS
LIN {X 0.233,Y -498.865,Z 1622.548,A 0.000,B 0.000,C 90.000,E1 98.568} C_DIS
LIN {X -0.133,Y -500.557,Z 1622.547,A 0.000,B 0.000,C 90.000,E1 98.398} C_DIS
LIN {X -0.207,Y -502.038,Z 1622.545,A 0.000,B 0.000,C 90.000,E1 98.163} C_DIS
LIN {X 0.216,Y -503.137,Z 1622.544,A 0.000,B 0.000,C 90.000,E1 97.871} C_DIS
LIN {X 0.012,Y -504.413,Z 1622.541,A 0.000,B 0.000,C 90.000,E1 97.409} C_DIS
LIN {X -0.185,Y -504.643,Z 1622.538,A 0.000,B 0.000,C 90.000,E1 96.947} C_DIS
LIN {X 0.125,Y -503.863,Z 1622.536,A 0.000,B 0.000,C 90.000,E1 96.429} C_DIS
LIN {X -0.063,Y -501.942,Z 1622.533,A 0.000,B 0.000,C 90.000,E1 95.967} C_DIS
LIN {X 0.192,Y -498.718,Z 1622.530,A 0.000,B 0.000,C 90.000,E1 95.454} C_DIS
LIN {X -0.154,Y -486.963,Z 1622.521,A 0.000,B 0.000,C 90.000,E1 93.784} C_DIS
LIN {X -0.126,Y -476.834,Z 1622.513,A 0.000,B 0.000,C 90.000,E1 92.293} C_DIS
LIN {X -0.071,Y -468.140,Z 1622.506,A 0.000,B 0.000,C 90.000,E1 91.031} C_DIS
LIN {X 0.091,Y -457.390,Z 1622.497,A 0.000,B 0.000,C 90.000,E1 89.484} C_DIS
LIN {X -0.149,Y -448.038,Z 1622.490,A 0.000,B 0.000,C 90.000,E1 88.224} C_DIS
LIN {X -0.057,Y -438.301,Z 1622.483,A 0.000,B 0.000,C 90.000,E1 86.906} C_DIS
LIN {X 0.053,Y -426.342,Z 1622.474,A 0.000,B 0.000,C 90.000,E1 85.298} C_DIS
LIN {X -0.208,Y -410.534,Z 1622.462,A 0.000,B 0.000,C 90.000,E1 83.166} C_DIS
LIN {X -0.155,Y -390.205,Z 1622.445,A 0.000,B 0.000,C 90.000,E1 80.095} C_DIS
LIN {X -0.165,Y -373.023,Z 1622.429,A 0.000,B 0.000,C 90.000,E1 77.229} C_DIS
LIN {X -0.117,Y -358.300,Z 1622.414,A 0.000,B 0.000,C 90.000,E1 74.574} C_DIS
LIN {X 0.054,Y -342.526,Z 1622.397,A 0.000,B 0.000,C 90.000,E1 71.529} C_DIS
LIN {X -0.069,Y -331.932,Z 1622.385,A 0.000,B 0.000,C 90.000,E1 69.390} C_DIS
LIN {X -0.035,Y -320.337,Z 1622.371,A 0.000,B 0.000,C 90.000,E1 66.869} C_DIS
LIN {X 0.047,Y -307.072,Z 1622.354,A 0.000,B 0.000,C 90.000,E1 63.640} C_DIS
LIN {X -0.160,Y -298.010,Z 1622.341,A 0.000,B 0.000,C 90.000,E1 61.385} C_DIS
LIN {X 0.134,Y -291.392,Z 1622.332,A 0.000,B 0.000,C 90.000,E1 59.665} C_DIS
LIN {X 0.046,Y -283.151,Z 1622.320,A 0.000,B 0.000,C 90.000,E1 57.661} C_DIS
LIN {X 0.007,Y -275.971,Z 1622.311,A 0.000,B 0.000,C 90.000,E1 55.960} C_DIS
LIN {X -0.058,Y -265.742,Z 1622.297,A 0.000,B 0.000,C 90.000,E1 53.543} C_DIS
LIN {X 0.029,Y -255.641,Z 1622.284,A 0.000,B 0.000,C 90.000,E1 51.045} C_DIS
LIN {X -0.016,Y -244.633,Z 1622.268,A 0.000,B 0.000,C 90.000,E1 48.162} C_DIS
LIN {X -0.041,Y -233.378,Z 1622.249,A 0.000,B 0.000,C 90.000,E1 44.838} C_DIS
LIN {X -0.041,Y -223.159,Z 1622.230,A 0.000,B 0.000,C 90.000,E1 41.434} C_DIS
LIN {X 0.015,Y -214.919,Z 1622.213,A 0.000,B 0.000,C 90.000,E1 38.338} C_DIS
LIN {X -0.084,Y -207.525,Z 1622.196,A 0.000,B 0.000,C 90.000,E1 35.231} C_DIS
LIN {X 0.068,Y -200.891,Z 1622.178,A 0.000,B 0.000,C 90.000,E1 32.005} C_DIS
LIN {X -0.085,Y -194.970,Z 1622.160,A 0.000,B 0.000,C 90.000,E1 28.821} C_DIS
LIN {X -0.049,Y -189.767,Z 1622.142,A 0.000,B 0.000,C 90.000,E1 25.540} C_DIS
LIN {X 0.034,Y -185.291,Z 1622.123,A 0.000,B 0.000,C 90.000,E1 22.206} C_DIS
LIN {X -0.065,Y -180.582,Z 1622.100,A 0.000,B 0.000,C 90.000,E1 18.055} C_DIS
LIN {X -0.060,Y -176.682,Z 1622.077,A 0.000,B 0.000,C 90.000,E1 13.828} C_DIS
LIN {X -0.033,Y -173.513,Z 1622.053,A 0.000,B 0.000,C 90.000,E1 9.557} C_DIS
LIN {X -0.075,Y -170.648,Z 1622.020,A 0.000,B 0.000,C 90.000,E1 3.555} C_DIS
LIN {X 0.026,Y -171.080,Z 1621.925,A 0.000,B 0.000,C 90.000,E1 346.533} C_DIS
LIN {X -0.079,Y -174.337,Z 1621.896,A 0.000,B 0.000,C 90.000,E1 341.402} C_DIS
LIN {X -0.061,Y -177.499,Z 1621.878,A 0.000,B 0.000,C 90.000,E1 337.975} C_DIS
LIN {X 0.078,Y -181.601,Z 1621.859,A 0.000,B 0.000,C 90.000,E1 334.537} C_DIS
LIN {X 0.066,Y -186.596,Z 1621.840,A 0.000,B 0.000,C 90.000,E1 331.179} C_DIS
LIN {X 0.031,Y -192.407,Z 1621.822,A 0.000,B 0.000,C 90.000,E1 327.867} C_DIS
LIN {X -0.040,Y -198.954,Z 1621.803,A 0.000,B 0.000,C 90.000,E1 324.609} C_DIS
LIN {X -0.035,Y -206.319,Z 1621.785,A 0.000,B 0.000,C 90.000,E1 321.376} C_DIS
LIN {X -0.083,Y -213.565,Z 1621.770,A 0.000,B 0.000,C 90.000,E1 318.609} C_DIS
LIN {X -0.080,Y -222.865,Z 1621.753,A 0.000,B 0.000,C 90.000,E1 315.486} C_DIS
LIN {X 0.009,Y -233.235,Z 1621.736,A 0.000,B 0.000,C 90.000,E1 312.405} C_DIS
LIN {X -0.047,Y -240.387,Z 1621.725,A 0.000,B 0.000,C 90.000,E1 310.539} C_DIS
LIN {X 0.039,Y -248.315,Z 1621.715,A 0.000,B 0.000,C 90.000,E1 308.669} C_DIS
LIN {X -0.033,Y -258.912,Z 1621.703,A 0.000,B 0.000,C 90.000,E1 306.503} C_DIS
LIN {X 0.074,Y -272.837,Z 1621.689,A 0.000,B 0.000,C 90.000,E1 303.992} C_DIS
LIN {X 0.011,Y -286.146,Z 1621.677,A 0.000,B 0.000,C 90.000,E1 301.926} C_DIS
LIN {X 0.174,Y -305.579,Z 1621.662,A 0.000,B 0.000,C 90.000,E1 299.205} C_DIS
LIN {X 0.132,Y -320.460,Z 1621.652,A 0.000,B 0.000,C 90.000,E1 297.257} C_DIS
LIN {X 0.124,Y -332.755,Z 1621.643,A 0.000,B 0.000,C 90.000,E1 295.668} C_DIS
LIN {X -0.009,Y -344.721,Z 1621.634,A 0.000,B 0.000,C 90.000,E1 294.131} C_DIS
LIN {X 0.123,Y -359.100,Z 1621.624,A 0.000,B 0.000,C 90.000,E1 292.280} C_DIS
LIN {X 0.201,Y -373.466,Z 1621.614,A 0.000,B 0.000,C 90.000,E1 290.482} C_DIS
LIN {X 0.034,Y -380.262,Z 1621.609,A 0.000,B 0.000,C 90.000,E1 289.631} C_DIS
LIN {X -0.084,Y -386.565,Z 1621.604,A 0.000,B 0.000,C 90.000,E1 288.779} C_DIS
LIN {X 0.232,Y -392.425,Z 1621.599,A 0.000,B 0.000,C 90.000,E1 287.873} C_DIS
LIN {X 0.107,Y -397.659,Z 1621.595,A 0.000,B 0.000,C 90.000,E1 287.040} C_DIS
LIN {X 0.036,Y -402.079,Z 1621.590,A 0.000,B 0.000,C 90.000,E1 286.205} C_DIS
LIN {X 0.002,Y -405.670,Z 1621.585,A 0.000,B 0.000,C 90.000,E1 285.371} C_DIS
LIN {X -0.098,Y -407.633,Z 1621.582,A 0.000,B 0.000,C 90.000,E1 284.828} C_DIS
LIN {X 0.099,Y -409.162,Z 1621.579,A 0.000,B 0.000,C 90.000,E1 284.245} C_DIS
LIN {X 0.012,Y -410.333,Z 1621.576,A 0.000,B 0.000,C 90.000,E1 283.703} C_DIS
LIN {X -0.167,Y -411.032,Z 1621.573,A 0.000,B 0.000,C 90.000,E1 283.175} C_DIS
LIN {X 0.064,Y -411.267,Z 1621.570,A 0.000,B 0.000,C 90.000,E1 282.591} C_DIS
LIN {X -0.102,Y -411.050,Z 1621.567,A 0.000,B 0.000,C 90.000,E1 282.063} C_DIS
LIN {X 0.136,Y -410.243,Z 1621.564,A 0.000,B 0.000,C 90.000,E1 281.478} C_DIS
LIN {X -0.029,Y -408.875,Z 1621.561,A 0.000,B 0.000,C 90.000,E1 280.950} C_DIS
LIN {X 0.200,Y -406.924,Z 1621.558,A 0.000,B 0.000,C 90.000,E1 280.366} C_DIS
LIN {X -0.051,Y -404.290,Z 1621.555,A 0.000,B 0.000,C 90.000,E1 279.849} C_DIS
LIN {X 0.148,Y -400.978,Z 1621.552,A 0.000,B 0.000,C 90.000,E1 279.265} C_DIS
LIN {X -0.130,Y -397.103,Z 1621.548,A 0.000,B 0.000,C 90.000,E1 278.746} C_DIS
LIN {X 0.025,Y -392.618,Z 1621.545,A 0.000,B 0.000,C 90.000,E1 278.163} C_DIS
LIN {X 0.174,Y -384.904,Z 1621.541,A 0.000,B 0.000,C 90.000,E1 277.296} C_DIS
LIN {X 0.012,Y -379.292,Z 1621.538,A 0.000,B 0.000,C 90.000,E1 276.777} C_DIS
LIN {X 0.085,Y -373.431,Z 1621.535,A 0.000,B 0.000,C 90.000,E1 276.258} C_DIS
LIN {X 0.011,Y -367.388,Z 1621.532,A 0.000,B 0.000,C 90.000,E1 275.796} C_DIS
LIN {X 0.171,Y -361.177,Z 1621.530,A 0.000,B 0.000,C 90.000,E1 275.334} C_DIS
LIN {X 0.076,Y -351.516,Z 1621.526,A 0.000,B 0.000,C 90.000,E1 274.759} C_DIS
LIN {X 0.031,Y -341.831,Z 1621.524,A 0.000,B 0.000,C 90.000,E1 274.245} C_DIS
LIN {X -0.029,Y -331.884,Z 1621.521,A 0.000,B 0.000,C 90.000,E1 273.784} C_DIS
LIN {X -0.087,Y -322.119,Z 1621.519,A 0.000,B 0.000,C 90.000,E1 273.383} C_DIS
LIN {X 0.093,Y -312.210,Z 1621.517,A 0.000,B 0.000,C 90.000,E1 272.980} C_DIS
LIN {X -0.123,Y -301.980,Z 1621.515,A 0.000,B 0.000,C 90.000,E1 272.694} C_DIS
LIN {X -0.055,Y -290.784,Z 1621.513,A 0.000,B 0.000,C 90.000,E1 272.407} C_DIS
LIN {X 0.042,Y -278.212,Z 1621.512,A 0.000,B 0.000,C 90.000,E1 272.178} C_DIS
LIN {X 0.120,Y -256.969,Z 1621.511,A 0.000,B 0.000,C 90.000,E1 271.949} C_DIS
LIN {X -0.019,Y -229.749,Z 1621.510,A 0.000,B 0.000,C 90.000,E1 271.776} C_DIS
LIN {X -0.018,Y -215.747,Z 1621.510,A 0.000,B 0.000,C 90.000,E1 271.718} C_DIS
LIN {X -0.058,Y -207.930,Z 1621.509,A 0.000,B 0.000,C 90.000,E1 271.718} C_DIS
LIN {X -0.087,Y -181.315,Z 1621.509,A 0.000,B 0.000,C 90.000,E1 271.718} C_DIS
LIN {X -0.087,Y -181.556,Z 1621.500,A 0.000,B 0.000,C 90.000,E1 270.000} C_DIS
LIN {X 0.080,Y -180.842,Z 1621.472,A 0.000,B 0.000,C 90.000,E1 264.894} C_DIS
LIN {X -0.018,Y -178.950,Z 1621.444,A 0.000,B 0.000,C 90.000,E1 259.859} C_DIS
LIN {X -0.001,Y -176.854,Z 1621.425,A 0.000,B 0.000,C 90.000,E1 256.464} C_DIS
LIN {X -0.029,Y -175.513,Z 1621.411,A 0.000,B 0.000,C 90.000,E1 253.921} C_DIS
LIN {X -0.027,Y -172.253,Z 1621.387,A 0.000,B 0.000,C 90.000,E1 249.645} C_DIS
LIN {X 0.012,Y -171.731,Z 1621.382,A 0.000,B 0.000,C 90.000,E1 248.773} C_DIS
LIN {X 0.020,Y -167.327,Z 1621.353,A 0.000,B 0.000,C 90.000,E1 243.589} C_DIS
LIN {X -0.048,Y -166.711,Z 1621.349,A 0.000,B 0.000,C 90.000,E1 242.743} C_DIS
LIN {X 0.090,Y -162.692,Z 1621.324,A 0.000,B 0.000,C 90.000,E1 238.329} C_DIS
LIN {X -0.072,Y -161.382,Z 1621.314,A 0.000,B 0.000,C 90.000,E1 236.628} C_DIS
LIN {X -0.029,Y -157.375,Z 1621.290,A 0.000,B 0.000,C 90.000,E1 232.190} C_DIS
LIN {X 0.006,Y -155.368,Z 1621.275,A 0.000,B 0.000,C 90.000,E1 229.504} C_DIS
LIN {X 0.052,Y -151.708,Z 1621.250,A 0.000,B 0.000,C 90.000,E1 225.000} C_DIS
LIN {X 0.063,Y -149.899,Z 1621.235,A 0.000,B 0.000,C 90.000,E1 222.285} C_DIS
LIN {X 0.086,Y -146.758,Z 1621.210,A 0.000,B 0.000,C 90.000,E1 217.729} C_DIS
LIN {X -0.016,Y -145.326,Z 1621.195,A 0.000,B 0.000,C 90.000,E1 215.025} C_DIS
LIN {X 0.025,Y -142.409,Z 1621.164,A 0.000,B 0.000,C 90.000,E1 209.489} C_DIS
LIN {X -0.050,Y -141.393,Z 1621.148,A 0.000,B 0.000,C 90.000,E1 206.744} C_DIS
LIN {X -0.061,Y -139.353,Z 1621.112,A 0.000,B 0.000,C 90.000,E1 200.248} C_DIS
LIN {X 0.059,Y -138.792,Z 1621.097,A 0.000,B 0.000,C 90.000,E1 197.402} C_DIS
LIN {X -0.019,Y -138.346,Z 1621.055,A 0.000,B 0.000,C 90.000,E1 189.962} C_DIS
LIN {X -0.002,Y -139.379,Z 1621.009,A 0.000,B 0.000,C 90.000,E1 181.547} C_DIS
LIN {X 0.052,Y -141.271,Z 1620.972,A 0.000,B 0.000,C 90.000,E1 175.008} C_DIS
LIN {X 0.010,Y -142.637,Z 1620.957,A 0.000,B 0.000,C 90.000,E1 172.243} C_DIS
LIN {X -0.039,Y -144.967,Z 1620.931,A 0.000,B 0.000,C 90.000,E1 167.645} C_DIS
LIN {X -0.048,Y -147.595,Z 1620.911,A 0.000,B 0.000,C 90.000,E1 163.976} C_DIS
LIN {X -0.018,Y -150.211,Z 1620.891,A 0.000,B 0.000,C 90.000,E1 160.315} C_DIS
LIN {X 0.049,Y -153.598,Z 1620.870,A 0.000,B 0.000,C 90.000,E1 156.666} C_DIS
LIN {X 0.036,Y -157.014,Z 1620.850,A 0.000,B 0.000,C 90.000,E1 153.076} C_DIS
LIN {X -0.031,Y -161.134,Z 1620.831,A 0.000,B 0.000,C 90.000,E1 149.537} C_DIS
LIN {X -0.086,Y -163.234,Z 1620.821,A 0.000,B 0.000,C 90.000,E1 147.788} C_DIS
LIN {X -0.083,Y -167.667,Z 1620.801,A 0.000,B 0.000,C 90.000,E1 144.276} C_DIS
LIN {X 0.066,Y -171.490,Z 1620.787,A 0.000,B 0.000,C 90.000,E1 141.618} C_DIS
LIN {X 0.110,Y -176.421,Z 1620.768,A 0.000,B 0.000,C 90.000,E1 138.162} C_DIS
LIN {X -0.019,Y -180.716,Z 1620.754,A 0.000,B 0.000,C 90.000,E1 135.648} C_DIS
LIN {X -0.038,Y -186.120,Z 1620.735,A 0.000,B 0.000,C 90.000,E1 132.285} C_DIS
LIN {X 0.021,Y -190.758,Z 1620.721,A 0.000,B 0.000,C 90.000,E1 129.769} C_DIS
LIN {X -0.071,Y -196.512,Z 1620.703,A 0.000,B 0.000,C 90.000,E1 126.503} C_DIS
LIN {X 0.006,Y -201.288,Z 1620.689,A 0.000,B 0.000,C 90.000,E1 124.040} C_DIS
LIN {X -0.036,Y -205.757,Z 1620.675,A 0.000,B 0.000,C 90.000,E1 121.592} C_DIS
LIN {X -0.109,Y -325.174,Z 1620.675,A 0.000,B 0.000,C 90.000,E1 121.592} C_DIS
LIN {X -0.039,Y -330.625,Z 1620.674,A 0.000,B 0.000,C 90.000,E1 121.386} C_DIS
LIN {X -0.086,Y -333.122,Z 1620.673,A 0.000,B 0.000,C 90.000,E1 121.209} C_DIS
LIN {X 0.167,Y -336.480,Z 1620.671,A 0.000,B 0.000,C 90.000,E1 120.797} C_DIS
LIN {X -0.071,Y -338.400,Z 1620.670,A 0.000,B 0.000,C 90.000,E1 120.541} C_DIS
LIN {X -0.138,Y -339.901,Z 1620.668,A 0.000,B 0.000,C 90.000,E1 120.256} C_DIS
LIN {X -0.081,Y -353.262,Z 1620.651,A 0.000,B 0.000,C 90.000,E1 117.180} C_DIS
LIN {X 0.024,Y -366.793,Z 1620.636,A 0.000,B 0.000,C 90.000,E1 114.463} C_DIS
LIN {X 0.115,Y -380.142,Z 1620.623,A 0.000,B 0.000,C 90.000,E1 112.099} C_DIS
